// TIA Portal project "ENSACADORA_V4_021024_OPTIMIZADO" (V18)

(* hardware
DEVICE "SIMATIC 1200 station_1"  S7-1200 Station
   slot 0: "S7-1200 rack"  S7-1200 Rack  Rack  V1.0
   slot 1: "Master"  CPU 1212C DC/DC/Rly  6ES7 212-1HE40-0XB0  V4.5
   slot 2: "DI 8x24VDC/DQ 8xRelay_1"  SM 1223 DI8/DQ8 x relay  6ES7 223-1PH32-0XB0  V2.0
   slot 3: "AQ 2x14BIT_1"  SM 1232 AQ2  6ES7 232-4HB32-0XB0  V2.1
   slot 101: "CM 1241 (RS422/485)_1"  6ES7 241-1CH32-0XB0  V2.2
*)

// ===== PLC "Master"  CPU 1212C DC/DC/Rly =====

VAR_GLOBAL   // PLC tag table "A_Bits_programa"
   "COM_ACTIVA" AT %M261.1 : Bool;
   "AUX_OUT_VIBRADOR_TIME" AT %M267.1 : Bool;
   "ABRIENDO_COMP_CARGA" AT %M267.0 : Bool;
   "AUX_TIME_VIBRADOR" AT %M266.7 : Bool;
   "ACTIVAR MOTOR" AT %M266.6 : Bool;
   "AUX_OUT_COMPUERTA_BARRIDO_ABIERTA" AT %M266.5 : Bool;
   "AUX_OUT_VIBRADOR_BARRIDO" AT %M266.4 : Bool;
   "AUX_OUT_MOTOR_BARRIDO" AT %M266.3 : Bool;
   "AUX_OUT_COMPUERTA_MANUAL" AT %M266.2 : Bool;
   "AUX_OUT_VIBRADOR_MANUAL" AT %M266.1 : Bool;
   "AUX_OUT_MOTOR_MANUAL" AT %M266.0 : Bool;
   "ZERO RES" AT %M265.7 : Bool;
   "AUX_HACER_ZERO" AT %M265.6 : Bool;
   "BAS_EN_ZERO" AT %M265.5 : Bool;
   "BAS_TARA_HECHA" AT %M265.4 : Bool;
   "BAS_OVERLOAD" AT %M265.3 : Bool;
   "BAS_UNDERLOAD" AT %M265.2 : Bool;
   "BAS_ESTABLE" AT %M265.1 : Bool;
   "PB_POLARIDAD" AT %M265.0 : Bool;
   "AUX_SENSOR_COMP_CARGA_ABIERTA" AT %M264.7 : Bool;
   "AUX_VAL_COMP_CARGA_ABIERTA" AT %M264.6 : Bool;
   "AUX_INICIAR_CICLO" AT %M264.5 : Bool;
   "AUX_ERROR_COM_BASCULA" AT %M264.4 : Bool;
   "AUX_RESET_CICLO" AT %M264.3 : Bool;
   "AUX_MODO_BARRIDO" AT %M264.2 : Bool;
   "AUX_MODO_AUTOMATICO" AT %M264.1 : Bool;
   "AUX_MODO_MANUAL" AT %M264.0 : Bool;
   "AUX_INICIAR_LLENADO" AT %M256.0 : Bool;
   "AUX_PARAR_LLENADO" AT %M256.1 : Bool;
   "AUX_PARO_EMERGENCIA" AT %M256.2 : Bool;
   "AUX_SENSOR_INICIO_COMPUERTA" AT %M256.3 : Bool;
   "AUX_SENSOR_FINAL_COMPUERTA" AT %M256.4 : Bool;
   "FirstScan_PREGUNTAR" AT %M50.0 : Bool;
   "SENTIDO_MOTOR" AT %M259.3 : Bool;
   "AUX_ZERO_MANUAL" AT %M260.6 : Bool;
   "FrmHmi_HacerZeroBas" AT %M260.7 : Bool;
   "FrmHmi_ResetFallas" AT %M261.0 : Bool;   // x
   "RESETEAR FALLAS" AT %M261.2 : Bool;
   "INCIAR_CICLO" AT %M262.0 : Bool;
   "APAGAR_CICLO" AT %M262.1 : Bool;
   "AUX_INPUT_SOBRECARGA_MOTOR" AT %M262.6 : Bool;
   "AUX_FALLA_ARRANQUE_VDF" AT %M256.5 : Bool;
   "AUX_FALLA_COMPUERTA_ABIERTA_DOSIFICAR" AT %M256.6 : Bool;
   "AUX_FALLA_VARIADOR" AT %M256.7 : Bool;
   "AUX_BLINK_TORRETA_AMARILLO_ON" AT %M259.4 : Bool;
   "AUX_BLINK_TORRETA_AMARILLO_OFF" AT %M259.5 : Bool;
   "AUX_BLINK_TORRETA_VERDE_ON" AT %M259.6 : Bool;
   "AUX_BLINK_TORRETA_VERDE_OFF" AT %M259.7 : Bool;
   "AUX_OUT_TORRETA_C_ROJO" AT %M262.2 : Bool;
   "AUX_OUT_TORRETA_C_AMARILLO" AT %M262.3 : Bool;
   "AUX_OUT_TORRETA_C_VERDE" AT %M262.4 : Bool;
   "AUX_OUT_TORRETA_BUZZER" AT %M262.5 : Bool;
   "TOLERANCIA DE PESO BASCULA" AT %M259.0 : Bool;
   "SET_INDICADOR_CAPACIDAD" AT %M252.0 : Bool;
   "FROM_HMI_LEER_CAPACIDAD" AT %M252.1 : Bool;
   "PARO EMERGENCIA" AT %M252.2 : Bool;
END_VAR

VAR_GLOBAL   // PLC tag table "A_Byte_programa"
   "STEP_COM" AT %MB257 : Byte;
END_VAR

VAR_GLOBAL   // PLC tag table "A_Word_programa"
   "Refe_Frec_FromHmi_ToVdf_PENDENTE" AT %MW0 : Int;
   "SETPOINT" AT %MW2 : Int;
   "ESTATUS_OPERACION" AT %MW8 : Int;
   "STEP_BASCULA" AT %MW10 : Int;
   "ESTATUS VARIADOR" AT %MW268 : Word;
END_VAR

VAR_GLOBAL   // PLC tag table "A_DWord_programa"
   "TARAR" AT %MD36 : Real;
   "PESO_NETO" AT %MD40 : Real;
   "PESO_NETO_BASCULA" AT %MD44 : Real;
   "MAYOR_QUE_SETPOINT" AT %MD48 : Real;
   "MENOR_QUE_SETPOINT" AT %MD52 : Real;
   "DIV" AT %MD20 : DWord;
   "FILTRO" AT %MD24 : DWord;
   "DIFERENCIA" AT %MD28 : DWord;
   "PUNTO DE CORTE" AT %MD32 : DWord;
   "DEFAULT CORTE SETPOINT" AT %MD4 : DWord;
   "TOLERANCIA DE PESO MAXIMO" AT %MD272 : DWord;
   "PESO NETO BASCULA ENTERO" AT %MD276 : DWord;
   "SALIDA REF FREC DIVIDA HMI" AT %MD280 : DWord;
   "SALIDA FREC DIVIDIDA HMI" AT %MD284 : DWord;
   "lectura resgistro bascula" AT %MD56 : UDInt;
   "SALIDA AMPERAJE" AT %MD60 : Real;
END_VAR

VAR_GLOBAL   // PLC tag table "B_Calibracion"
   "ENVIAR_PESO_A_CALIBRAR" AT %M271.7 : Bool;
   "CONFIRMAR_PESO_CALIBRAR" AT %M271.6 : Bool;
   "CANCELAR_CALIBRACION" AT %M271.5 : Bool;
   "GUARDAR_CALIBRACION" AT %M271.4 : Bool;
   "CAPTURAR_PESO_BASCULA" AT %M271.3 : Bool;
   "CAPTURAR_ZERO_BASCULA" AT %M271.2 : Bool;
   "RESET_INDICADOR" AT %M271.1 : Bool;
   "VER_CALIBRACION" AT %M271.0 : Bool;
   "PESO_PARA_CALIBRAR" AT %MD92 : DInt;
END_VAR

VAR_GLOBAL   // PLC tag table "C_Fallas"
   "TIEMPO_APAGADO_VIBRADOR" AT %MD16 : DInt;
   "TIEMPO_ENCENDIDO_VIBRADOR" AT %MD12 : DInt;
   "Falla sobrecarga motor" AT %M270.7 : Bool;
   "Falla subcarga bascula" AT %M270.6 : Bool;
   "Falla sobrecarga bascula" AT %M270.5 : Bool;
   "FALLA_NO_SE_PUEDE_INICIAR_EN_ZERO" AT %M270.4 : Bool;
   "Fallas activas" AT %M270.3 : Bool;
   "Falla en el tiempo de vibrador" AT %M270.2 : Bool;
   "Falla al abrir compuerta descarga" AT %M270.1 : Bool;
   "Falla al cerrar compuerta descarga" AT %M270.0 : Bool;
   "TIMER_FALLAS_ON" AT %M259.2 : Bool;
   "TIMER_FALLAS_OFF" AT %M259.1 : Bool;
   "ERROR_MODBUS" AT %M267.2 : Bool;
   "AUX_ERROR_MODBUS" AT %M267.3 : Bool;
   "ERROR_VARIADOR" AT %M267.4 : Bool;
   "AUX_ERROR_VARIADOR" AT %M267.5 : Bool;
   "ERROR AL ENCENDER EL VARIADOR" AT %M267.6 : Bool;
   "FALLA AL ENCENDER EL MOTOR CON LA COMPUERTA CERRADA" AT %M267.7 : Bool;
END_VAR

VAR_GLOBAL   // PLC tag table "D_Entradas"
   "Input_SensorInicioPistonComp" AT %I0.4 : Bool;
   "Input_IniciarLLenado" AT %I0.0 : Bool;
   "Input_ParoEmergencia" AT %I0.2 : Bool;
   "Input_PararLLenado" AT %I0.1 : Bool;
   "Input_Sobrecarga_motor" AT %I0.3 : Bool;
   "Input_SensorFinPistonComp" AT %I0.5 : Bool;
END_VAR

VAR_GLOBAL   // PLC tag table "D_Salidas"
   "OUT_COMPUERTA_ABIERTA" AT %Q0.0 : Bool;
   "OUT_VIBRADOR" AT %Q0.1 : Bool;
   "TORRETA_C_ROJO" AT %Q0.3 : Bool;
   "TORRETA_C_AMARILLO" AT %Q0.4 : Bool;
   "TORRETA_C_VERDE" AT %Q0.5 : Bool;
   "TORRETA_BUZZER" AT %Q0.2 : Bool;
   "Kg_To_CCM" AT %QW112 : Word;
END_VAR

VAR_GLOBAL   // PLC tag table "E_Hmi"
   "FrmHmi_Barrido" AT %M263.4 : Bool;
   "FrmHmi_DesactivarModBarrido" AT %M263.3 : Bool;
   "FrmHmi_ActivarModBarrido" AT %M263.2 : Bool;
   "FrmHmi_Automatico" AT %M263.1 : Bool;
   "FrmHmi_ModManual" AT %M263.0 : Bool;
   "FrmHmi_ApagarVibradorEnsacadora" AT %M260.5 : Bool;
   "FrmHmi_EncenderVibradorEnsacadora" AT %M260.4 : Bool;
   "FrmHmi_DesactivarPistonCompuerta" AT %M260.3 : Bool;
   "FrmHmi_ActivarPistonCompuerta" AT %M260.2 : Bool;
   "FrmHmi_ApagarMotorHelicoidal" AT %M260.1 : Bool;
   "FrmHmi_EncenderMotorHelicoidal" AT %M260.0 : Bool;
END_VAR

TYPE "typeModbusCommLoad"
VERSION : 0.1
   STRUCT
      done : Bool := FALSE;
      error : Bool := FALSE;
      status : Word := W#16#0;
      errorStatus : Word := W#16#0;
      doneStored : Bool := FALSE;
   END_STRUCT;
END_TYPE

TYPE "typeModbusMaster"
VERSION : 0.1
   STRUCT
      req : Bool := FALSE;
      mbAddr : UInt;
      mode : USInt := 0;
      dataAddr : UDInt := 0;
      dataLen : UInt := 0;
      done : Bool := FALSE;
      busy : Bool := FALSE;
      error : Bool := FALSE;
      status : Word := W#16#0;
      errorStatus : Word := W#16#0;
   END_STRUCT;
END_TYPE

TYPE "typeDataPtr"
VERSION : 0.1
   STRUCT
      data : Array[0..11] of Int;
   END_STRUCT;
END_TYPE

TYPE "typeModbusVariador"
   STRUCT
      req : Bool := FALSE;
      mbAddr : UInt := 0;
      mode : USInt := 0;
      dataAddr : UDInt := 0;
      dataLen : UInt := 0;
      done : Bool := FALSE;
      busy : Bool := FALSE;
      error : Bool := FALSE;
      status : Word;
      errorStatus : Word;
   END_STRUCT;
END_TYPE

DATA_BLOCK "MasterData"   // DB1
{ S7_Optimized_Access := 'FALSE' }
VERSION : 0.1
   VAR
      "WRITE BASCULA" : Array[0..3] of Int;
      "READ BASCULA" : Array[0..10] of Int;
      "STATUS CAL" : Array[0..9] of Int;
      "WRITE VDF MOTOR" : Array[0..1] of Int;
      "READ VDF MOTOR" : Array[0..10] of Int;
      "PESO CALIBRAR" : Array[0..1] of Int;
      "LEER PESO CALIBRAR" : Array[0..2] of Int;
      "CAPACIDAD INDICADOR" : Array[0..1] of Int;
   END_VAR
BEGIN
END_DATA_BLOCK

DATA_BLOCK "Process"   // DB3
{ S7_Optimized_Access := 'TRUE' }
VERSION : 0.1
   VAR
      "step" : USInt := 1;
      edge : Bool := false;
      modbusMaster : "typeModbusMaster";
      modbusCommLoad : "typeModbusCommLoad";
   END_VAR
BEGIN
   modbusMaster.mbAddr := 2;
   modbusMaster.dataLen := 2;
END_DATA_BLOCK

DATA_BLOCK "HACER TARA_DB"   // DB6
{ S7_Optimized_Access := 'TRUE' }
VERSION : 0.1
// stored: InstanceOfName HACER TARA
"HACER TARA"
BEGIN
END_DATA_BLOCK

DATA_BLOCK "PORCENTAJE DE CORTE VDF GRUESO_DB_DB"   // DB9
{ S7_Optimized_Access := 'TRUE' }
VERSION : 0.1
// stored: InstanceOfName PORCENTAJE DE CORTE VDF GRUESO_DB
"PORCENTAJE DE CORTE VDF GRUESO_DB"
BEGIN
END_DATA_BLOCK

DATA_BLOCK "HACER TARA_DB_1"   // DB11
{ S7_Optimized_Access := 'TRUE' }
VERSION : 0.1
// stored: InstanceOfName HACER TARA
"HACER TARA"
BEGIN
END_DATA_BLOCK

DATA_BLOCK "db_variador"   // DB27
{ S7_Optimized_Access := 'TRUE' }
VERSION : 0.1
   VAR
      modbusVariador : "typeModbusVariador";
   END_VAR
BEGIN
END_DATA_BLOCK

// folder: System blocks/Program resources

DATA_BLOCK "IEC_Timer_0_DB"   // DB2
{ S7_Optimized_Access := 'TRUE' }
AUTHOR : Simatic
FAMILY : IEC
NAME : IEC_TMR
VERSION : 1.0
// stored: InstanceOfName IEC_TIMER
"IEC_TIMER"
BEGIN
END_DATA_BLOCK

DATA_BLOCK "IEC_Timer_0_DB_1"   // DB7
{ S7_Optimized_Access := 'TRUE' }
AUTHOR : Simatic
FAMILY : IEC
NAME : IEC_TMR
VERSION : 1.0
// stored: InstanceOfName IEC_TIMER
"IEC_TIMER"
BEGIN
END_DATA_BLOCK

DATA_BLOCK "IEC_Timer_0_DB_2"   // DB8
{ S7_Optimized_Access := 'TRUE' }
AUTHOR : Simatic
FAMILY : IEC
NAME : IEC_TMR
VERSION : 1.0
// stored: InstanceOfName IEC_TIMER
"IEC_TIMER"
BEGIN
END_DATA_BLOCK

DATA_BLOCK "IEC_Timer_0_DB_3"   // DB10
{ S7_Optimized_Access := 'TRUE' }
AUTHOR : Simatic
FAMILY : IEC
NAME : IEC_TMR
VERSION : 1.0
// stored: InstanceOfName IEC_TIMER
"IEC_TIMER"
BEGIN
END_DATA_BLOCK

DATA_BLOCK "IEC_Timer_0_DB_4"   // DB12
{ S7_Optimized_Access := 'TRUE' }
AUTHOR : Simatic
FAMILY : IEC
NAME : IEC_TMR
VERSION : 1.0
// stored: InstanceOfName IEC_TIMER
"IEC_TIMER"
BEGIN
END_DATA_BLOCK

DATA_BLOCK "IEC_Timer_0_DB_5"   // DB13
{ S7_Optimized_Access := 'TRUE' }
AUTHOR : Simatic
FAMILY : IEC
NAME : IEC_TMR
VERSION : 1.0
// stored: InstanceOfName IEC_TIMER
"IEC_TIMER"
BEGIN
END_DATA_BLOCK

DATA_BLOCK "IEC_Timer_0_DB_6"   // DB14
{ S7_Optimized_Access := 'TRUE' }
AUTHOR : Simatic
FAMILY : IEC
NAME : IEC_TMR
VERSION : 1.0
// stored: InstanceOfName IEC_TIMER
"IEC_TIMER"
BEGIN
END_DATA_BLOCK

DATA_BLOCK "IEC_Timer_0_DB_7"   // DB15
{ S7_Optimized_Access := 'TRUE' }
AUTHOR : Simatic
FAMILY : IEC
NAME : IEC_TMR
VERSION : 1.0
// stored: InstanceOfName IEC_TIMER
"IEC_TIMER"
BEGIN
END_DATA_BLOCK

DATA_BLOCK "IEC_Timer_0_DB_8"   // DB16
{ S7_Optimized_Access := 'TRUE' }
AUTHOR : Simatic
FAMILY : IEC
NAME : IEC_TMR
VERSION : 1.0
// stored: InstanceOfName IEC_TIMER
"IEC_TIMER"
BEGIN
END_DATA_BLOCK

DATA_BLOCK "IEC_Timer_0_DB_9"   // DB17
{ S7_Optimized_Access := 'TRUE' }
AUTHOR : Simatic
FAMILY : IEC
NAME : IEC_TMR
VERSION : 1.0
// stored: InstanceOfName IEC_TIMER
"IEC_TIMER"
BEGIN
END_DATA_BLOCK

DATA_BLOCK "IEC_Timer_0_DB_10"   // DB18
{ S7_Optimized_Access := 'TRUE' }
AUTHOR : Simatic
FAMILY : IEC
NAME : IEC_TMR
VERSION : 1.0
// stored: InstanceOfName IEC_TIMER
"IEC_TIMER"
BEGIN
END_DATA_BLOCK

DATA_BLOCK "IEC_Timer_0_DB_11"   // DB19
{ S7_Optimized_Access := 'TRUE' }
AUTHOR : Simatic
FAMILY : IEC
NAME : IEC_TMR
VERSION : 1.0
// stored: InstanceOfName IEC_TIMER
"IEC_TIMER"
BEGIN
END_DATA_BLOCK

DATA_BLOCK "IEC_Timer_0_DB_17"   // DB20
{ S7_Optimized_Access := 'TRUE' }
AUTHOR : Simatic
FAMILY : IEC
NAME : IEC_TMR
VERSION : 1.0
// stored: InstanceOfName IEC_TIMER
"IEC_TIMER"
BEGIN
END_DATA_BLOCK

DATA_BLOCK "IEC_Timer_0_DB_12"   // DB21
{ S7_Optimized_Access := 'TRUE' }
AUTHOR : Simatic
FAMILY : IEC
NAME : IEC_TMR
VERSION : 1.0
// stored: InstanceOfName IEC_TIMER
"IEC_TIMER"
BEGIN
END_DATA_BLOCK

DATA_BLOCK "IEC_Timer_0_DB_13"   // DB22
{ S7_Optimized_Access := 'TRUE' }
AUTHOR : Simatic
FAMILY : IEC
NAME : IEC_TMR
VERSION : 1.0
// stored: InstanceOfName IEC_TIMER
"IEC_TIMER"
BEGIN
END_DATA_BLOCK

DATA_BLOCK "IEC_Timer_0_DB_19"   // DB23
{ S7_Optimized_Access := 'TRUE' }
AUTHOR : Simatic
FAMILY : IEC
NAME : IEC_TMR
VERSION : 1.0
// stored: InstanceOfName IEC_TIMER
"IEC_TIMER"
BEGIN
END_DATA_BLOCK

DATA_BLOCK "IEC_Timer_0_DB_14"   // DB24
{ S7_Optimized_Access := 'TRUE' }
AUTHOR : Simatic
FAMILY : IEC
NAME : IEC_TMR
VERSION : 1.0
// stored: InstanceOfName IEC_TIMER
"IEC_TIMER"
BEGIN
END_DATA_BLOCK

DATA_BLOCK "IEC_Timer_0_DB_15"   // DB25
{ S7_Optimized_Access := 'TRUE' }
AUTHOR : Simatic
FAMILY : IEC
NAME : IEC_TMR
VERSION : 1.0
// stored: InstanceOfName IEC_TIMER
"IEC_TIMER"
BEGIN
END_DATA_BLOCK

DATA_BLOCK "IEC_Timer_0_DB_16"   // DB26
{ S7_Optimized_Access := 'TRUE' }
AUTHOR : Simatic
FAMILY : IEC
NAME : IEC_TMR
VERSION : 1.0
// stored: InstanceOfName IEC_TIMER
"IEC_TIMER"
BEGIN
END_DATA_BLOCK

DATA_BLOCK "IEC_Timer_0_DB_18"   // DB28
{ S7_Optimized_Access := 'TRUE' }
AUTHOR : Simatic
FAMILY : IEC
NAME : IEC_TMR
VERSION : 1.0
// stored: InstanceOfName IEC_TIMER
"IEC_TIMER"
BEGIN
END_DATA_BLOCK

DATA_BLOCK "IEC_Timer_0_DB_20"   // DB29
{ S7_Optimized_Access := 'TRUE' }
AUTHOR : Simatic
FAMILY : IEC
NAME : IEC_TMR
VERSION : 1.0
// stored: InstanceOfName IEC_TIMER
"IEC_TIMER"
BEGIN
END_DATA_BLOCK

// folder: (top level)

FUNCTION_BLOCK "HACER TARA"   // FB1, LAD
{ S7_Optimized_Access := 'TRUE' }
VERSION : 0.1
   VAR_INPUT
      TARAR2 : Bool;
      TARAR1 : Bool;
   END_VAR
   VAR_OUTPUT
      "PESO NETO TARA" : Real;
   END_VAR
   VAR_TEMP
      TARA : Real;
      TA : Bool;
      TA2 : Bool;
      available : Bool;
   END_VAR
   VAR_TEMP   // added for the SCL form of the ladder/FBD networks
      _w1 : Bool;
   END_VAR
BEGIN

REGION Network 1
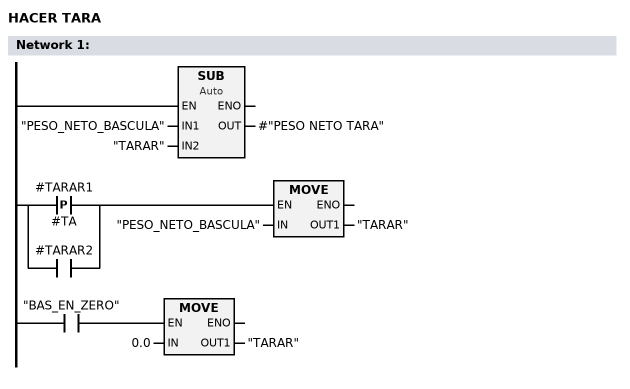
   RUNG wire#powerrail
      Sub(in1 := "PESO_NETO_BASCULA", in2 := "TARAR", out => #"PESO NETO TARA")
   END_RUNG
   RUNG wire#powerrail
      P_Contact(operand := #TARAR1, bit := #TA)
      wire#w1
      Move(in := "PESO_NETO_BASCULA", out1 => "TARAR")
   END_RUNG
   RUNG wire#powerrail
      Contact( #TARAR2 )
   END_RUNG wire#w1
   RUNG wire#powerrail
      Contact( "BAS_EN_ZERO" )
      Move(in := 0.0, out1 => "TARAR")
   END_RUNG
   // the same network as SCL:
   #"PESO NETO TARA" := "PESO_NETO_BASCULA" - "TARAR";
   #_w1 := #TARAR1 AND NOT #TA;   // rising edge of #TARAR1
   #TA := #TARAR1;
   IF #_w1 OR #TARAR2 THEN "TARAR" := "PESO_NETO_BASCULA"; END_IF;
   IF "BAS_EN_ZERO" THEN "TARAR" := 0.0; END_IF;
END_REGION
END_FUNCTION_BLOCK

FUNCTION_BLOCK "PORCENTAJE DE CORTE VDF GRUESO_DB"   // FB2, LAD
{ S7_Optimized_Access := 'TRUE' }
VERSION : 0.1
   VAR_INPUT
      "Set point" : Int;
      "% De Corte" : Int;
      PesoNeto : Real;
   END_VAR
   VAR_OUTPUT
      "Cantidad a cortar" : Real;
      "Bit OFF VDF Grueso" : Bool;
   END_VAR
   VAR_TEMP
      MULTI : Int;
   END_VAR
BEGIN

REGION Network 1
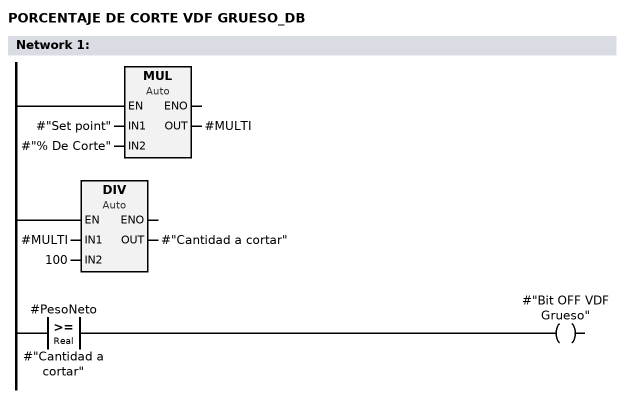
   RUNG wire#powerrail
      Mul(in1 := #"Set point", in2 := #"% De Corte", out => #MULTI)
   END_RUNG
   RUNG wire#powerrail
      Div(in1 := #MULTI, in2 := 100, out => #"Cantidad a cortar")
   END_RUNG
   RUNG wire#powerrail
      { S7_Templates := "SrcType := Real" } GE_Contact(in1 := #PesoNeto, in2 := #"Cantidad a cortar")
      Coil( #"Bit OFF VDF Grueso" )
   END_RUNG
   // the same network as SCL:
   #MULTI := #"Set point" * #"% De Corte";
   #"Cantidad a cortar" := #MULTI / 100;
   #"Bit OFF VDF Grueso" := #PesoNeto >= #"Cantidad a cortar";
END_REGION
END_FUNCTION_BLOCK

ORGANIZATION_BLOCK "1- COMUNICACION MODBUS"   // OB1, LAD, ProgramCycle
{ S7_Optimized_Access := 'TRUE' }
VERSION : 0.1
   VAR_INPUT
      Initial_Call : Bool;
      Remanence : Bool;
   END_VAR
   VAR_TEMP
      OutFrecMot : Int;
      OutRefFrecMot : Int;
      OutCorrienteMot : Real;
      "Bits Bascula" : DInt;
      "eroor com" : Bool;
      "weig neto" : Real;
      frecuencia : DInt;
   END_VAR
   VAR_TEMP   // added for the SCL form of the ladder/FBD networks
      _w1 : Bool;
   END_VAR
BEGIN

REGION Network 1: INICIALIZAR COMUNICACION
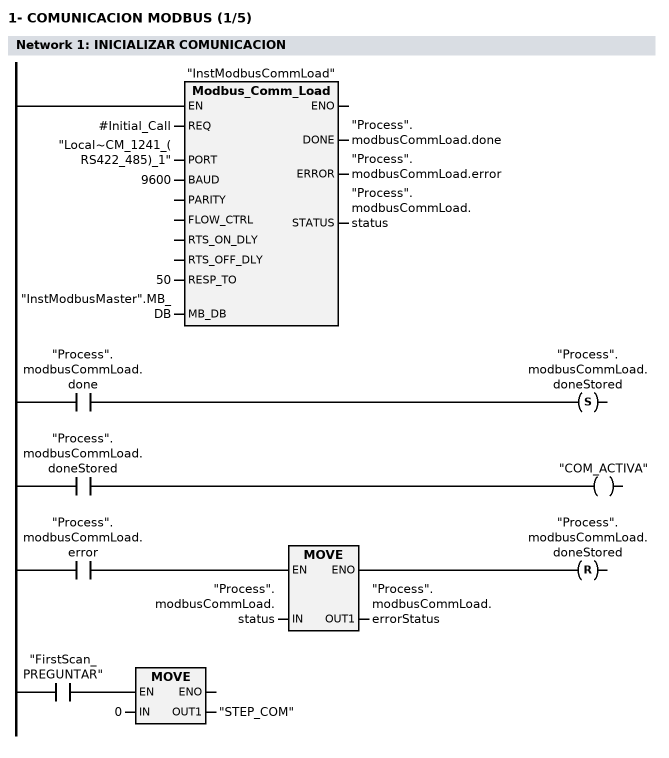
   // ENO of a box is taken as its EN; it also drops when the box reports an error
   "InstModbusCommLoad"(REQ := #Initial_Call,   // Modbus_Comm_Load
                        PORT := "Local~CM_1241_(RS422_485)_1",
                        BAUD := 9600,
                        RESP_TO := 50,
                        MB_DB := "InstModbusMaster".MB_DB,
                        DONE => "Process".modbusCommLoad.done,
                        ERROR => "Process".modbusCommLoad.error,
                        STATUS => "Process".modbusCommLoad.status);
   IF "Process".modbusCommLoad.done THEN "Process".modbusCommLoad.doneStored := TRUE; END_IF;
   "COM_ACTIVA" := "Process".modbusCommLoad.doneStored;
   IF "Process".modbusCommLoad.error THEN
       "Process".modbusCommLoad.errorStatus := "Process".modbusCommLoad.status;
       "Process".modbusCommLoad.doneStored := FALSE;
   END_IF;
   IF "FirstScan_PREGUNTAR" THEN "STEP_COM" := 0; END_IF;
END_REGION

REGION Network 2: LEER--ESCRIBIR, BASCULA
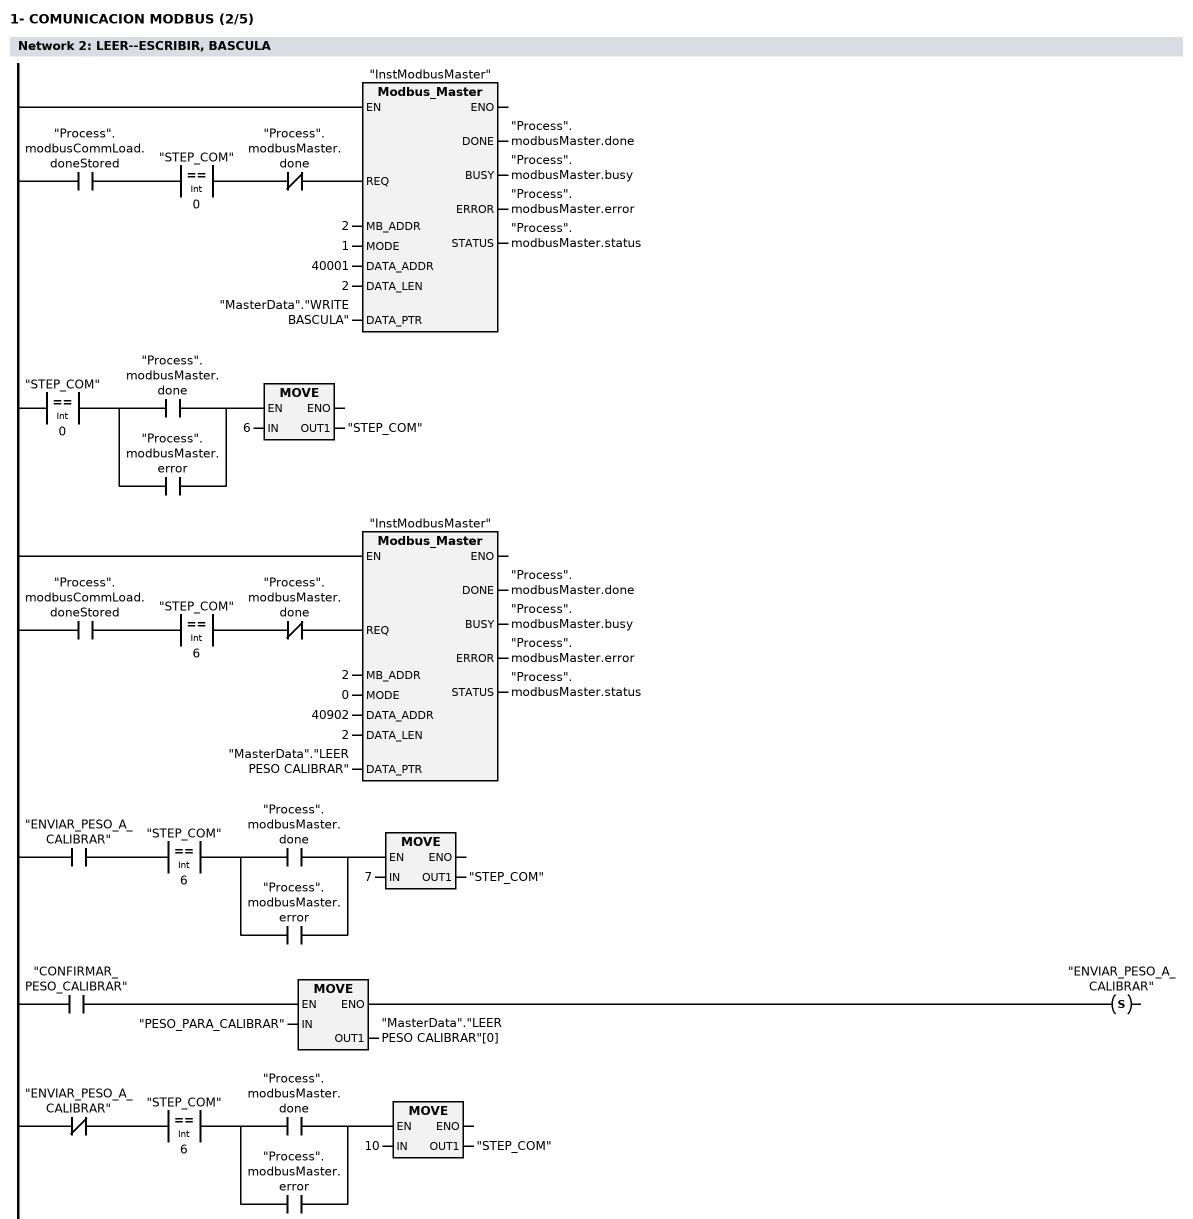
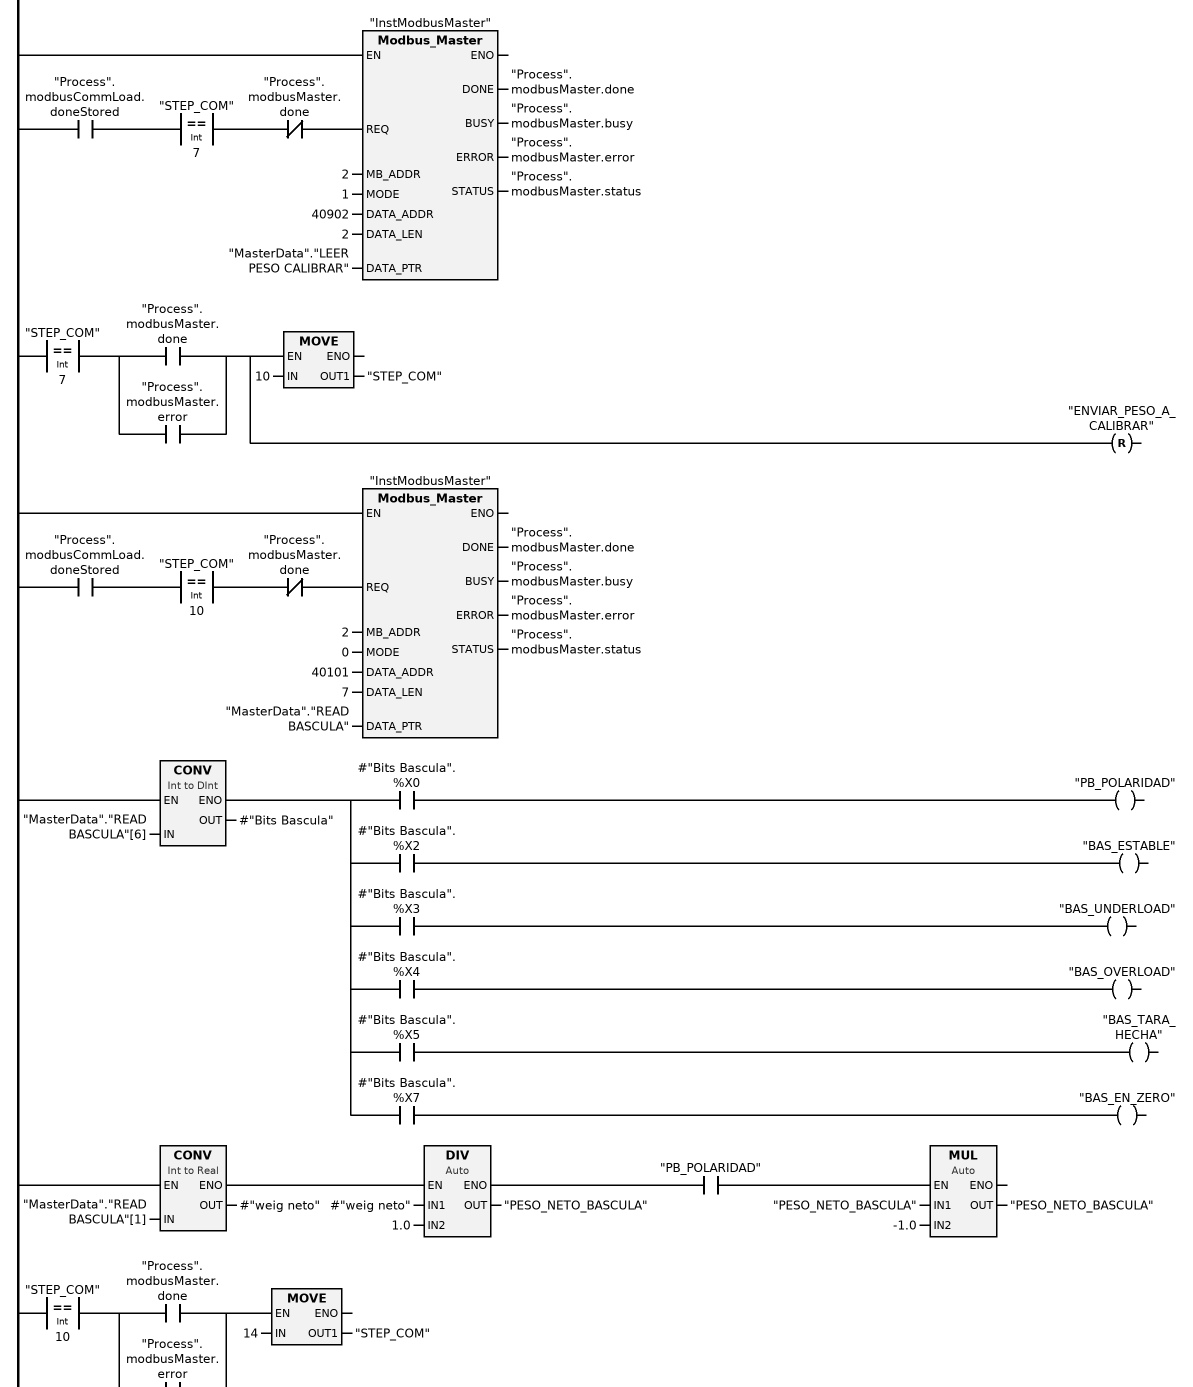
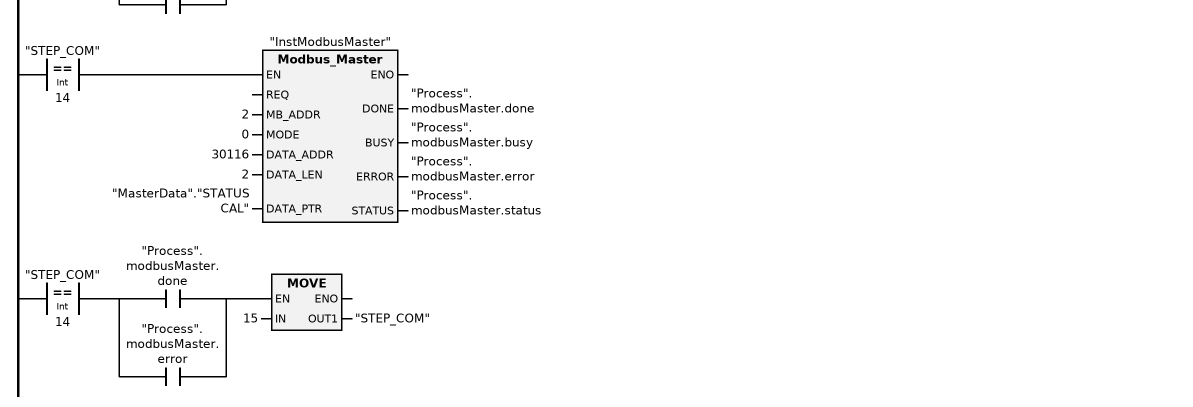
   "InstModbusMaster"(REQ := "Process".modbusCommLoad.doneStored AND ("STEP_COM" = 0) AND NOT "Process".modbusMaster.done,   // Modbus_Master
                      MB_ADDR := 2,
                      MODE := 1,
                      DATA_ADDR := 40001,
                      DATA_LEN := 2,
                      DATA_PTR := "MasterData"."WRITE BASCULA",
                      DONE => "Process".modbusMaster.done,
                      BUSY => "Process".modbusMaster.busy,
                      ERROR => "Process".modbusMaster.error,
                      STATUS => "Process".modbusMaster.status);
   IF ("STEP_COM" = 0) AND ("Process".modbusMaster.done OR "Process".modbusMaster.error) THEN
       "STEP_COM" := 6;
   END_IF;
   "InstModbusMaster"(REQ := "Process".modbusCommLoad.doneStored AND ("STEP_COM" = 6) AND NOT "Process".modbusMaster.done,   // Modbus_Master
                      MB_ADDR := 2,
                      MODE := 0,
                      DATA_ADDR := 40902,
                      DATA_LEN := 2,
                      DATA_PTR := "MasterData"."LEER PESO CALIBRAR",
                      DONE => "Process".modbusMaster.done,
                      BUSY => "Process".modbusMaster.busy,
                      ERROR => "Process".modbusMaster.error,
                      STATUS => "Process".modbusMaster.status);
   IF "ENVIAR_PESO_A_CALIBRAR" AND ("STEP_COM" = 6) AND ("Process".modbusMaster.done OR "Process".modbusMaster.error) THEN
       "STEP_COM" := 7;
   END_IF;
   IF "CONFIRMAR_PESO_CALIBRAR" THEN
       "MasterData"."LEER PESO CALIBRAR"[0] := "PESO_PARA_CALIBRAR";
       "ENVIAR_PESO_A_CALIBRAR" := TRUE;
   END_IF;
   IF NOT "ENVIAR_PESO_A_CALIBRAR" AND ("STEP_COM" = 6) AND ("Process".modbusMaster.done OR "Process".modbusMaster.error) THEN
       "STEP_COM" := 10;
   END_IF;
   "InstModbusMaster"(REQ := "Process".modbusCommLoad.doneStored AND ("STEP_COM" = 7) AND NOT "Process".modbusMaster.done,   // Modbus_Master
                      MB_ADDR := 2,
                      MODE := 1,
                      DATA_ADDR := 40902,
                      DATA_LEN := 2,
                      DATA_PTR := "MasterData"."LEER PESO CALIBRAR",
                      DONE => "Process".modbusMaster.done,
                      BUSY => "Process".modbusMaster.busy,
                      ERROR => "Process".modbusMaster.error,
                      STATUS => "Process".modbusMaster.status);
   #_w1 := ("STEP_COM" = 7) AND ("Process".modbusMaster.done OR "Process".modbusMaster.error);
   IF #_w1 THEN
       "STEP_COM" := 10;
       "ENVIAR_PESO_A_CALIBRAR" := FALSE;
   END_IF;
   "InstModbusMaster"(REQ := "Process".modbusCommLoad.doneStored AND ("STEP_COM" = 10) AND NOT "Process".modbusMaster.done,   // Modbus_Master
                      MB_ADDR := 2,
                      MODE := 0,
                      DATA_ADDR := 40101,
                      DATA_LEN := 7,
                      DATA_PTR := "MasterData"."READ BASCULA",
                      DONE => "Process".modbusMaster.done,
                      BUSY => "Process".modbusMaster.busy,
                      ERROR => "Process".modbusMaster.error,
                      STATUS => "Process".modbusMaster.status);
   #"Bits Bascula" := INT_TO_DINT("MasterData"."READ BASCULA"[6]);
   "PB_POLARIDAD" := #"Bits Bascula".%X0;
   "BAS_ESTABLE" := #"Bits Bascula".%X2;
   "BAS_UNDERLOAD" := #"Bits Bascula".%X3;
   "BAS_OVERLOAD" := #"Bits Bascula".%X4;
   "BAS_TARA_HECHA" := #"Bits Bascula".%X5;
   "BAS_EN_ZERO" := #"Bits Bascula".%X7;
   #"weig neto" := INT_TO_REAL("MasterData"."READ BASCULA"[1]);
   "PESO_NETO_BASCULA" := #"weig neto" / 1.0;
   IF "PB_POLARIDAD" THEN "PESO_NETO_BASCULA" := "PESO_NETO_BASCULA" * (-1.0); END_IF;
   IF ("STEP_COM" = 10) AND ("Process".modbusMaster.done OR "Process".modbusMaster.error) THEN
       "STEP_COM" := 14;
   END_IF;
   IF "STEP_COM" = 14 THEN
       "InstModbusMaster"(MB_ADDR := 2,   // Modbus_Master
                          MODE := 0,
                          DATA_ADDR := 30116,
                          DATA_LEN := 2,
                          DATA_PTR := "MasterData"."STATUS CAL",
                          DONE => "Process".modbusMaster.done,
                          BUSY => "Process".modbusMaster.busy,
                          ERROR => "Process".modbusMaster.error,
                          STATUS => "Process".modbusMaster.status);
   END_IF;
   IF ("STEP_COM" = 14) AND ("Process".modbusMaster.done OR "Process".modbusMaster.error) THEN
       "STEP_COM" := 15;
   END_IF;
END_REGION

REGION Network 3: FALLA EN LA BASCULA
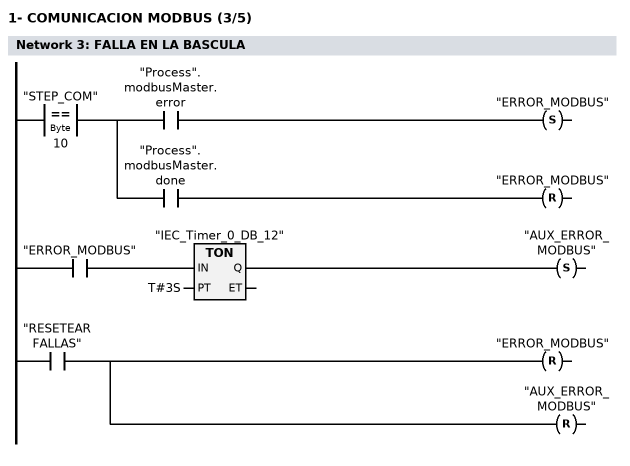
   #_w1 := "STEP_COM" = 10;
   IF #_w1 AND "Process".modbusMaster.error THEN "ERROR_MODBUS" := TRUE; END_IF;
   IF #_w1 AND "Process".modbusMaster.done THEN "ERROR_MODBUS" := FALSE; END_IF;
   "IEC_Timer_0_DB_12".TON(IN := "ERROR_MODBUS", PT := T#3S);
   IF "IEC_Timer_0_DB_12".Q THEN "AUX_ERROR_MODBUS" := TRUE; END_IF;
   IF "RESETEAR FALLAS" THEN
       "ERROR_MODBUS" := FALSE;
       "AUX_ERROR_MODBUS" := FALSE;
   END_IF;
END_REGION

REGION Network 4: LEER--ESCRIBIR, VDF MOTOR
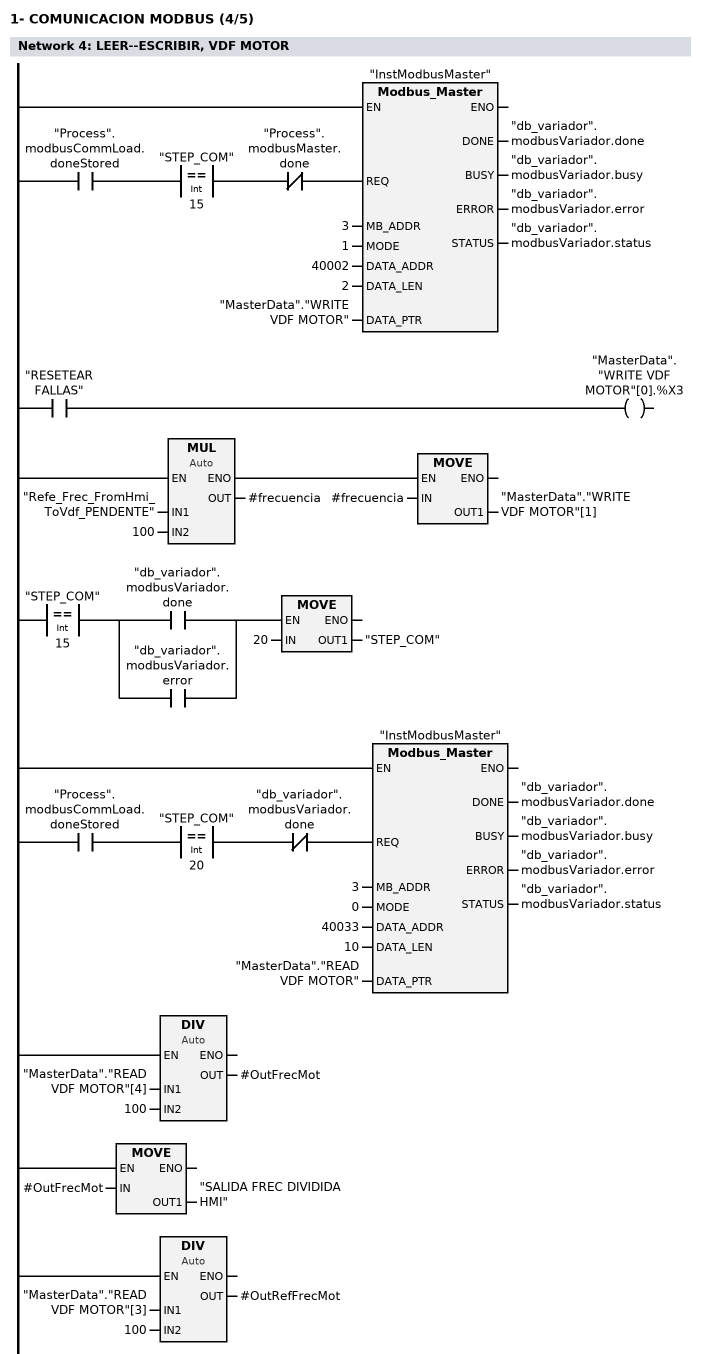
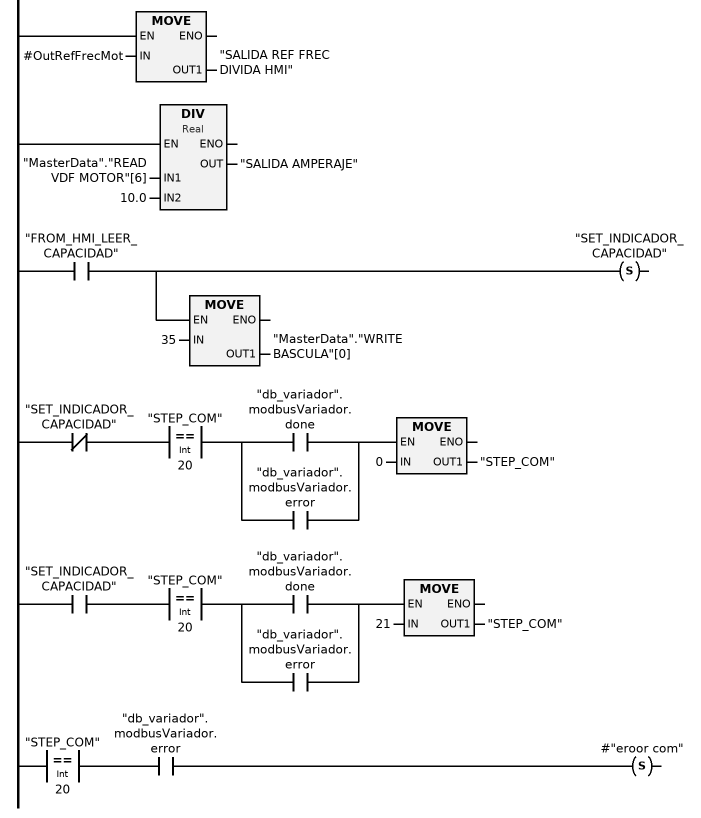
   "InstModbusMaster"(REQ := "Process".modbusCommLoad.doneStored AND ("STEP_COM" = 15) AND NOT "Process".modbusMaster.done,   // Modbus_Master
                      MB_ADDR := 3,
                      MODE := 1,
                      DATA_ADDR := 40002,
                      DATA_LEN := 2,
                      DATA_PTR := "MasterData"."WRITE VDF MOTOR",
                      DONE => "db_variador".modbusVariador.done,
                      BUSY => "db_variador".modbusVariador.busy,
                      ERROR => "db_variador".modbusVariador.error,
                      STATUS => "db_variador".modbusVariador.status);
   "MasterData"."WRITE VDF MOTOR"[0].%X3 := "RESETEAR FALLAS";
   #frecuencia := "Refe_Frec_FromHmi_ToVdf_PENDENTE" * 100;
   "MasterData"."WRITE VDF MOTOR"[1] := #frecuencia;
   IF ("STEP_COM" = 15) AND ("db_variador".modbusVariador.done OR "db_variador".modbusVariador.error) THEN
       "STEP_COM" := 20;
   END_IF;
   "InstModbusMaster"(REQ := "Process".modbusCommLoad.doneStored AND ("STEP_COM" = 20) AND NOT "db_variador".modbusVariador.done,   // Modbus_Master
                      MB_ADDR := 3,
                      MODE := 0,
                      DATA_ADDR := 40033,
                      DATA_LEN := 10,
                      DATA_PTR := "MasterData"."READ VDF MOTOR",
                      DONE => "db_variador".modbusVariador.done,
                      BUSY => "db_variador".modbusVariador.busy,
                      ERROR => "db_variador".modbusVariador.error,
                      STATUS => "db_variador".modbusVariador.status);
   #OutFrecMot := "MasterData"."READ VDF MOTOR"[4] / 100;
   "SALIDA FREC DIVIDIDA HMI" := #OutFrecMot;
   #OutRefFrecMot := "MasterData"."READ VDF MOTOR"[3] / 100;
   "SALIDA REF FREC DIVIDA HMI" := #OutRefFrecMot;
   "SALIDA AMPERAJE" := "MasterData"."READ VDF MOTOR"[6] / 10.0;
   IF "FROM_HMI_LEER_CAPACIDAD" THEN
       "SET_INDICADOR_CAPACIDAD" := TRUE;
       "MasterData"."WRITE BASCULA"[0] := 35;
   END_IF;
   IF NOT "SET_INDICADOR_CAPACIDAD" AND ("STEP_COM" = 20) AND ("db_variador".modbusVariador.done OR "db_variador".modbusVariador.error) THEN
       "STEP_COM" := 0;
   END_IF;
   IF "SET_INDICADOR_CAPACIDAD" AND ("STEP_COM" = 20) AND ("db_variador".modbusVariador.done OR "db_variador".modbusVariador.error) THEN
       "STEP_COM" := 21;
   END_IF;
   IF ("STEP_COM" = 20) AND "db_variador".modbusVariador.error THEN #"eroor com" := TRUE; END_IF;
END_REGION

REGION Network 5: LEER CAPACIDA DE BASCULA PARA CONVERSION 4MA-20MA A CMM
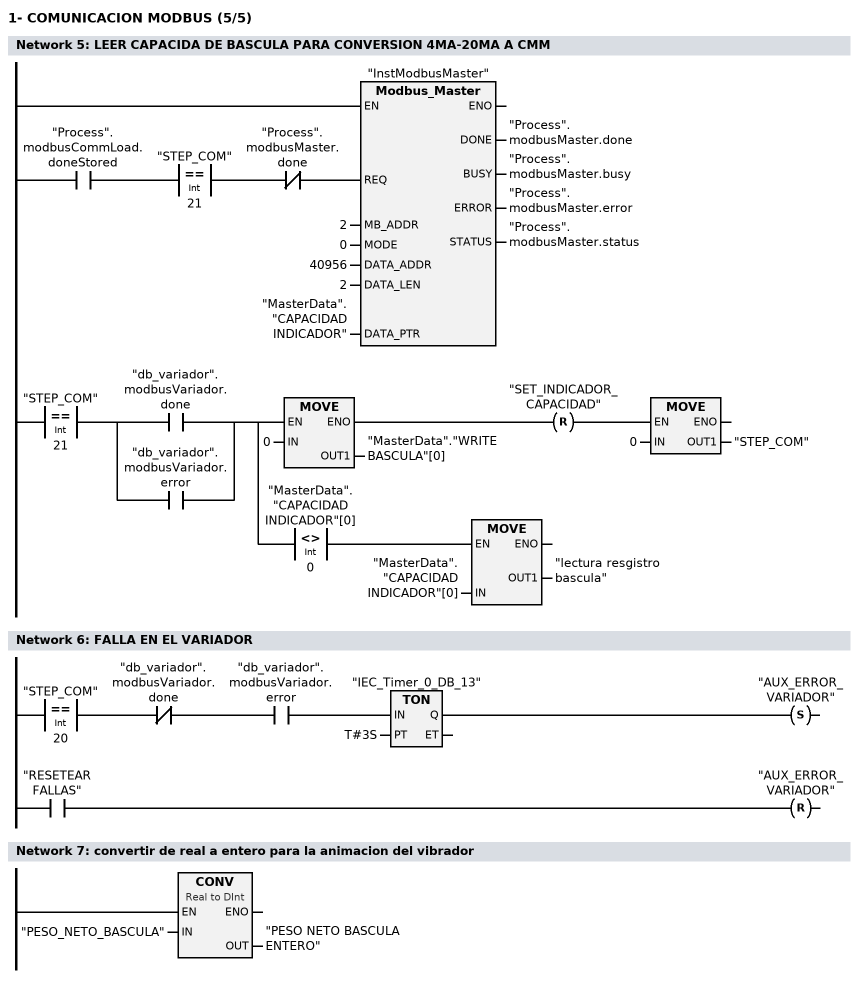
   "InstModbusMaster"(REQ := "Process".modbusCommLoad.doneStored AND ("STEP_COM" = 21) AND NOT "Process".modbusMaster.done,   // Modbus_Master
                      MB_ADDR := 2,
                      MODE := 0,
                      DATA_ADDR := 40956,
                      DATA_LEN := 2,
                      DATA_PTR := "MasterData"."CAPACIDAD INDICADOR",
                      DONE => "Process".modbusMaster.done,
                      BUSY => "Process".modbusMaster.busy,
                      ERROR => "Process".modbusMaster.error,
                      STATUS => "Process".modbusMaster.status);
   #_w1 := ("STEP_COM" = 21) AND ("db_variador".modbusVariador.done OR "db_variador".modbusVariador.error);
   IF #_w1 THEN
       "MasterData"."WRITE BASCULA"[0] := 0;
       "SET_INDICADOR_CAPACIDAD" := FALSE;
       "STEP_COM" := 0;
   END_IF;
   IF #_w1 AND ("MasterData"."CAPACIDAD INDICADOR"[0] <> 0) THEN
       "lectura resgistro bascula" := "MasterData"."CAPACIDAD INDICADOR"[0];
   END_IF;
END_REGION

REGION Network 6: FALLA EN EL VARIADOR
   "IEC_Timer_0_DB_13".TON(IN := ("STEP_COM" = 20) AND NOT "db_variador".modbusVariador.done AND "db_variador".modbusVariador.error,
                           PT := T#3S);
   IF "IEC_Timer_0_DB_13".Q THEN "AUX_ERROR_VARIADOR" := TRUE; END_IF;
   IF "RESETEAR FALLAS" THEN "AUX_ERROR_VARIADOR" := FALSE; END_IF;
END_REGION

REGION Network 7: convertir de real a entero para la animacion del vibrador
   RUNG wire#powerrail
      { S7_Templates := "[SrcType := Real, DestType := DInt]" } Convert(in := "PESO_NETO_BASCULA", out => "PESO NETO BASCULA ENTERO")
   END_RUNG
   // the same network as SCL:
   "PESO NETO BASCULA ENTERO" := REAL_TO_DINT("PESO_NETO_BASCULA");
END_REGION
END_ORGANIZATION_BLOCK

ORGANIZATION_BLOCK "2- ENTRADAS"   // OB123, LAD, ProgramCycle
{ S7_Optimized_Access := 'TRUE' }
VERSION : 0.1
   VAR_INPUT
      Initial_Call : Bool;
      Remanence : Bool;
   END_VAR
BEGIN

REGION Network 1: ENTRADAS FÍSICAS
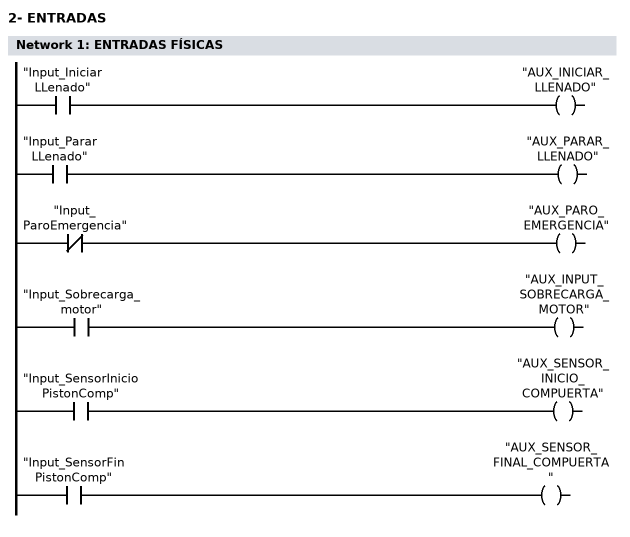
   RUNG wire#powerrail
      Contact( "Input_IniciarLLenado" )
      Coil( "AUX_INICIAR_LLENADO" )
   END_RUNG
   RUNG wire#powerrail
      Contact( "Input_PararLLenado" )
      Coil( "AUX_PARAR_LLENADO" )
   END_RUNG
   RUNG wire#powerrail
      I_Contact( "Input_ParoEmergencia" )
      Coil( "AUX_PARO_EMERGENCIA" )
   END_RUNG
   RUNG wire#powerrail
      Contact( "Input_Sobrecarga_motor" )
      Coil( "AUX_INPUT_SOBRECARGA_MOTOR" )
   END_RUNG
   RUNG wire#powerrail
      Contact( "Input_SensorInicioPistonComp" )
      Coil( "AUX_SENSOR_INICIO_COMPUERTA" )
   END_RUNG
   RUNG wire#powerrail
      Contact( "Input_SensorFinPistonComp" )
      Coil( "AUX_SENSOR_FINAL_COMPUERTA" )
   END_RUNG
   // the same network as SCL:
   "AUX_INICIAR_LLENADO" := "Input_IniciarLLenado";
   "AUX_PARAR_LLENADO" := "Input_PararLLenado";
   "AUX_PARO_EMERGENCIA" := NOT "Input_ParoEmergencia";
   "AUX_INPUT_SOBRECARGA_MOTOR" := "Input_Sobrecarga_motor";
   "AUX_SENSOR_INICIO_COMPUERTA" := "Input_SensorInicioPistonComp";
   "AUX_SENSOR_FINAL_COMPUERTA" := "Input_SensorFinPistonComp";
END_REGION
END_ORGANIZATION_BLOCK

ORGANIZATION_BLOCK "3- LOGICA LLENADO"   // OB124, LAD, ProgramCycle
{ S7_Optimized_Access := 'TRUE' }
VERSION : 0.1
   VAR_INPUT
      Initial_Call : Bool;
      Remanence : Bool;
   END_VAR
   VAR_TEMP
      inhabilitar : Bool;
      AVAILABLE : Bool;
      frecoMOT : Int;
      "TIME ENCENDIDO" : Time;
      "TIME APAGADO" : Time;
      "RESULTADO ENCENDIDO" : Int;
      "RESULTADO APAGADO" : Int;
      status_operacion : Bool;
   END_VAR
   VAR_TEMP   // added for the SCL form of the ladder/FBD networks
      _w1 : Bool;
      _w2 : Bool;
   END_VAR
BEGIN

REGION Network 1: MODO MANUAL, AUTOMATICO, BARRIDO
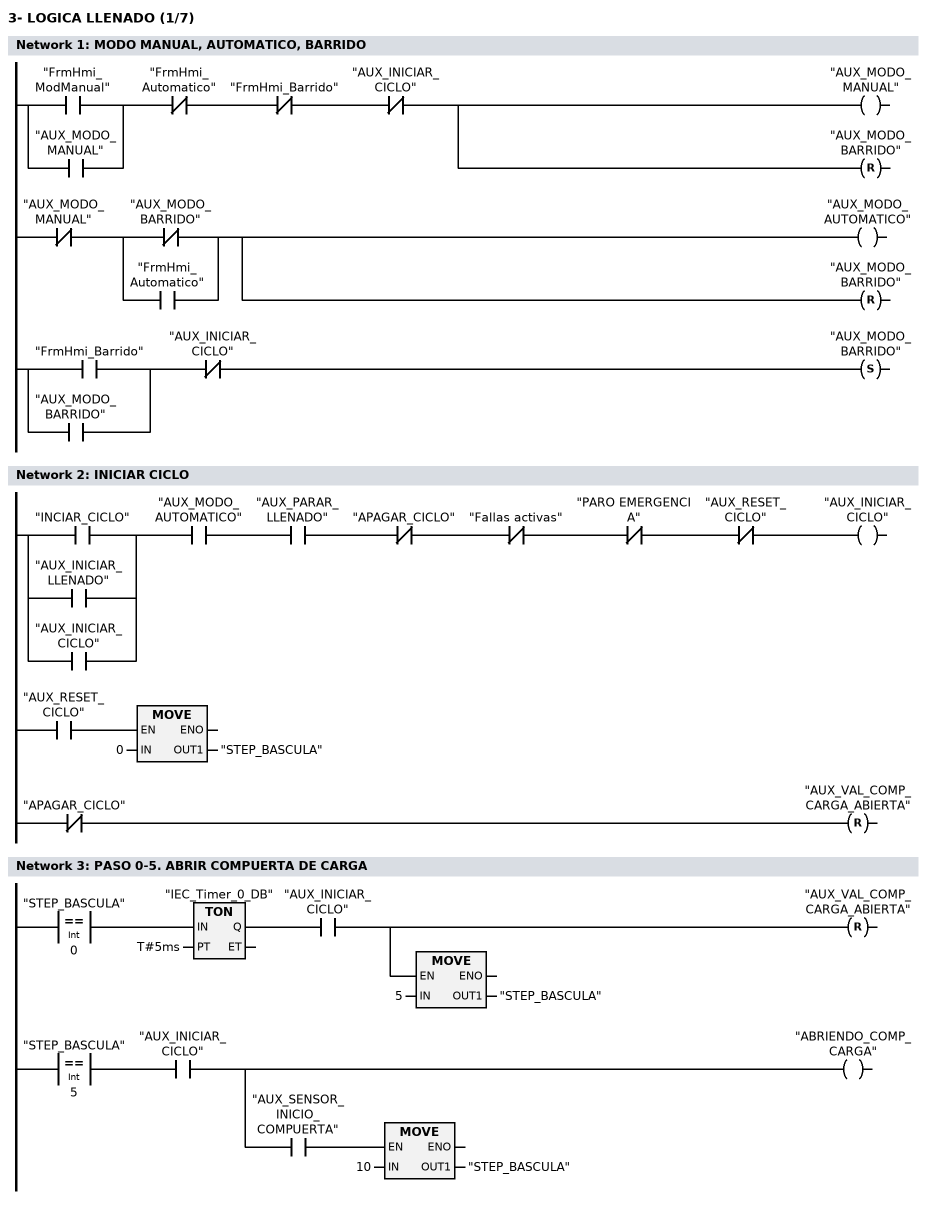
   RUNG wire#powerrail
      Contact( "FrmHmi_ModManual" )
      wire#w1
      I_Contact( "FrmHmi_Automatico" )
      I_Contact( "FrmHmi_Barrido" )
      I_Contact( "AUX_INICIAR_CICLO" )
      wire#w2
      Coil( "AUX_MODO_MANUAL" )
   END_RUNG
   RUNG wire#powerrail
      Contact( "AUX_MODO_MANUAL" )
   END_RUNG wire#w1
   RUNG wire#w2
      R_Coil( "AUX_MODO_BARRIDO" )
   END_RUNG
   RUNG wire#powerrail
      I_Contact( "AUX_MODO_MANUAL" )
      wire#w3
      I_Contact( "AUX_MODO_BARRIDO" )
      wire#w4
      Coil( "AUX_MODO_AUTOMATICO" )
   END_RUNG
   RUNG wire#w3
      Contact( "FrmHmi_Automatico" )
   END_RUNG wire#w4
   RUNG wire#w4
      R_Coil( "AUX_MODO_BARRIDO" )
   END_RUNG
   RUNG wire#powerrail
      Contact( "FrmHmi_Barrido" )
      wire#w5
      I_Contact( "AUX_INICIAR_CICLO" )
      S_Coil( "AUX_MODO_BARRIDO" )
   END_RUNG
   RUNG wire#powerrail
      Contact( "AUX_MODO_BARRIDO" )
   END_RUNG wire#w5
   // the same network as SCL:
   "AUX_MODO_MANUAL" := ("FrmHmi_ModManual" OR "AUX_MODO_MANUAL") AND NOT "FrmHmi_Automatico" AND NOT "FrmHmi_Barrido" AND NOT "AUX_INICIAR_CICLO";
   IF "AUX_MODO_MANUAL" THEN "AUX_MODO_BARRIDO" := FALSE; END_IF;
   "AUX_MODO_AUTOMATICO" := NOT "AUX_MODO_MANUAL" AND (NOT "AUX_MODO_BARRIDO" OR "FrmHmi_Automatico");
   IF "AUX_MODO_AUTOMATICO" THEN "AUX_MODO_BARRIDO" := FALSE; END_IF;
   IF ("FrmHmi_Barrido" OR "AUX_MODO_BARRIDO") AND NOT "AUX_INICIAR_CICLO" THEN
       "AUX_MODO_BARRIDO" := TRUE;
   END_IF;
END_REGION

REGION Network 2: INICIAR CICLO
   RUNG wire#powerrail
      Contact( "INCIAR_CICLO" )
      wire#w1
      Contact( "AUX_MODO_AUTOMATICO" )
      Contact( "AUX_PARAR_LLENADO" )
      I_Contact( "APAGAR_CICLO" )
      I_Contact( "Fallas activas" )
      I_Contact( "PARO EMERGENCIA" )
      I_Contact( "AUX_RESET_CICLO" )
      Coil( "AUX_INICIAR_CICLO" )
   END_RUNG
   RUNG wire#powerrail
      Contact( "AUX_INICIAR_LLENADO" )
   END_RUNG wire#w1
   RUNG wire#powerrail
      Contact( "AUX_INICIAR_CICLO" )
   END_RUNG wire#w1
   RUNG wire#powerrail
      Contact( "AUX_RESET_CICLO" )
      Move(in := 0, out1 => "STEP_BASCULA")
   END_RUNG
   RUNG wire#powerrail
      I_Contact( "APAGAR_CICLO" )
      R_Coil( "AUX_VAL_COMP_CARGA_ABIERTA" )
   END_RUNG
   // the same network as SCL:
   "AUX_INICIAR_CICLO" := ("INCIAR_CICLO" OR "AUX_INICIAR_LLENADO" OR "AUX_INICIAR_CICLO") AND "AUX_MODO_AUTOMATICO" AND "AUX_PARAR_LLENADO" AND NOT "APAGAR_CICLO" AND NOT "Fallas activas" AND NOT "PARO EMERGENCIA" AND NOT "AUX_RESET_CICLO";
   IF "AUX_RESET_CICLO" THEN "STEP_BASCULA" := 0; END_IF;
   IF NOT "APAGAR_CICLO" THEN "AUX_VAL_COMP_CARGA_ABIERTA" := FALSE; END_IF;
END_REGION

REGION Network 3: PASO 0-5. ABRIR COMPUERTA DE CARGA
   "IEC_Timer_0_DB".TON(IN := "STEP_BASCULA" = 0, PT := T#5ms);
   IF "IEC_Timer_0_DB".Q AND "AUX_INICIAR_CICLO" THEN
       "AUX_VAL_COMP_CARGA_ABIERTA" := FALSE;
       "STEP_BASCULA" := 5;
   END_IF;
   "ABRIENDO_COMP_CARGA" := ("STEP_BASCULA" = 5) AND "AUX_INICIAR_CICLO";
   IF "ABRIENDO_COMP_CARGA" AND "AUX_SENSOR_INICIO_COMPUERTA" THEN "STEP_BASCULA" := 10; END_IF;
END_REGION

REGION Network 4: PASO 10. HACER TARA
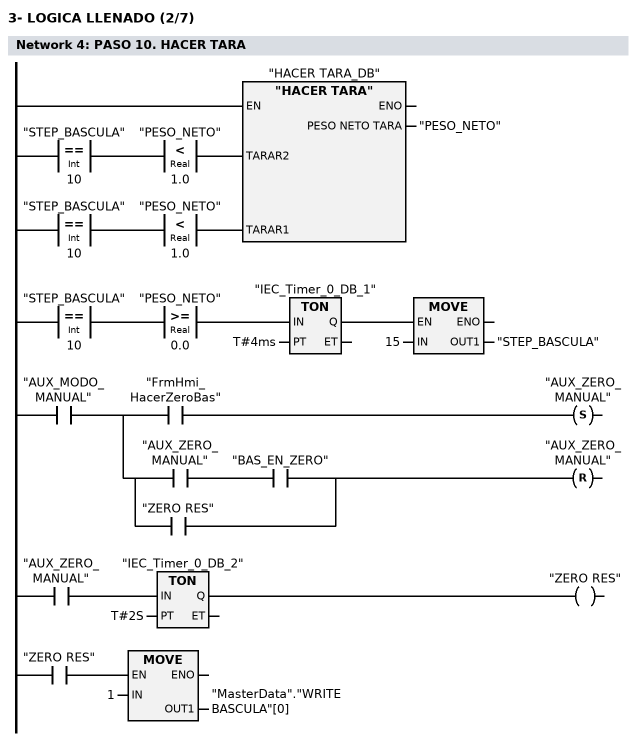
   "HACER TARA_DB"(TARAR2 := ("STEP_BASCULA" = 10) AND ("PESO_NETO" < 1.0),   // "HACER TARA"
                   TARAR1 := ("STEP_BASCULA" = 10) AND ("PESO_NETO" < 1.0),
                   "PESO NETO TARA" => "PESO_NETO");
   "IEC_Timer_0_DB_1".TON(IN := ("STEP_BASCULA" = 10) AND ("PESO_NETO" >= 0.0), PT := T#4ms);
   IF "IEC_Timer_0_DB_1".Q THEN "STEP_BASCULA" := 15; END_IF;
   IF "AUX_MODO_MANUAL" AND "FrmHmi_HacerZeroBas" THEN "AUX_ZERO_MANUAL" := TRUE; END_IF;
   IF "AUX_MODO_MANUAL" AND (("AUX_ZERO_MANUAL" AND "BAS_EN_ZERO") OR "ZERO RES") THEN
       "AUX_ZERO_MANUAL" := FALSE;
   END_IF;
   "IEC_Timer_0_DB_2".TON(IN := "AUX_ZERO_MANUAL", PT := T#2S);
   "ZERO RES" := "IEC_Timer_0_DB_2".Q;
   IF "ZERO RES" THEN "MasterData"."WRITE BASCULA"[0] := 1; END_IF;
END_REGION

REGION Network 5: PASO 15. ENCENDER Y APAGAR MOTORES
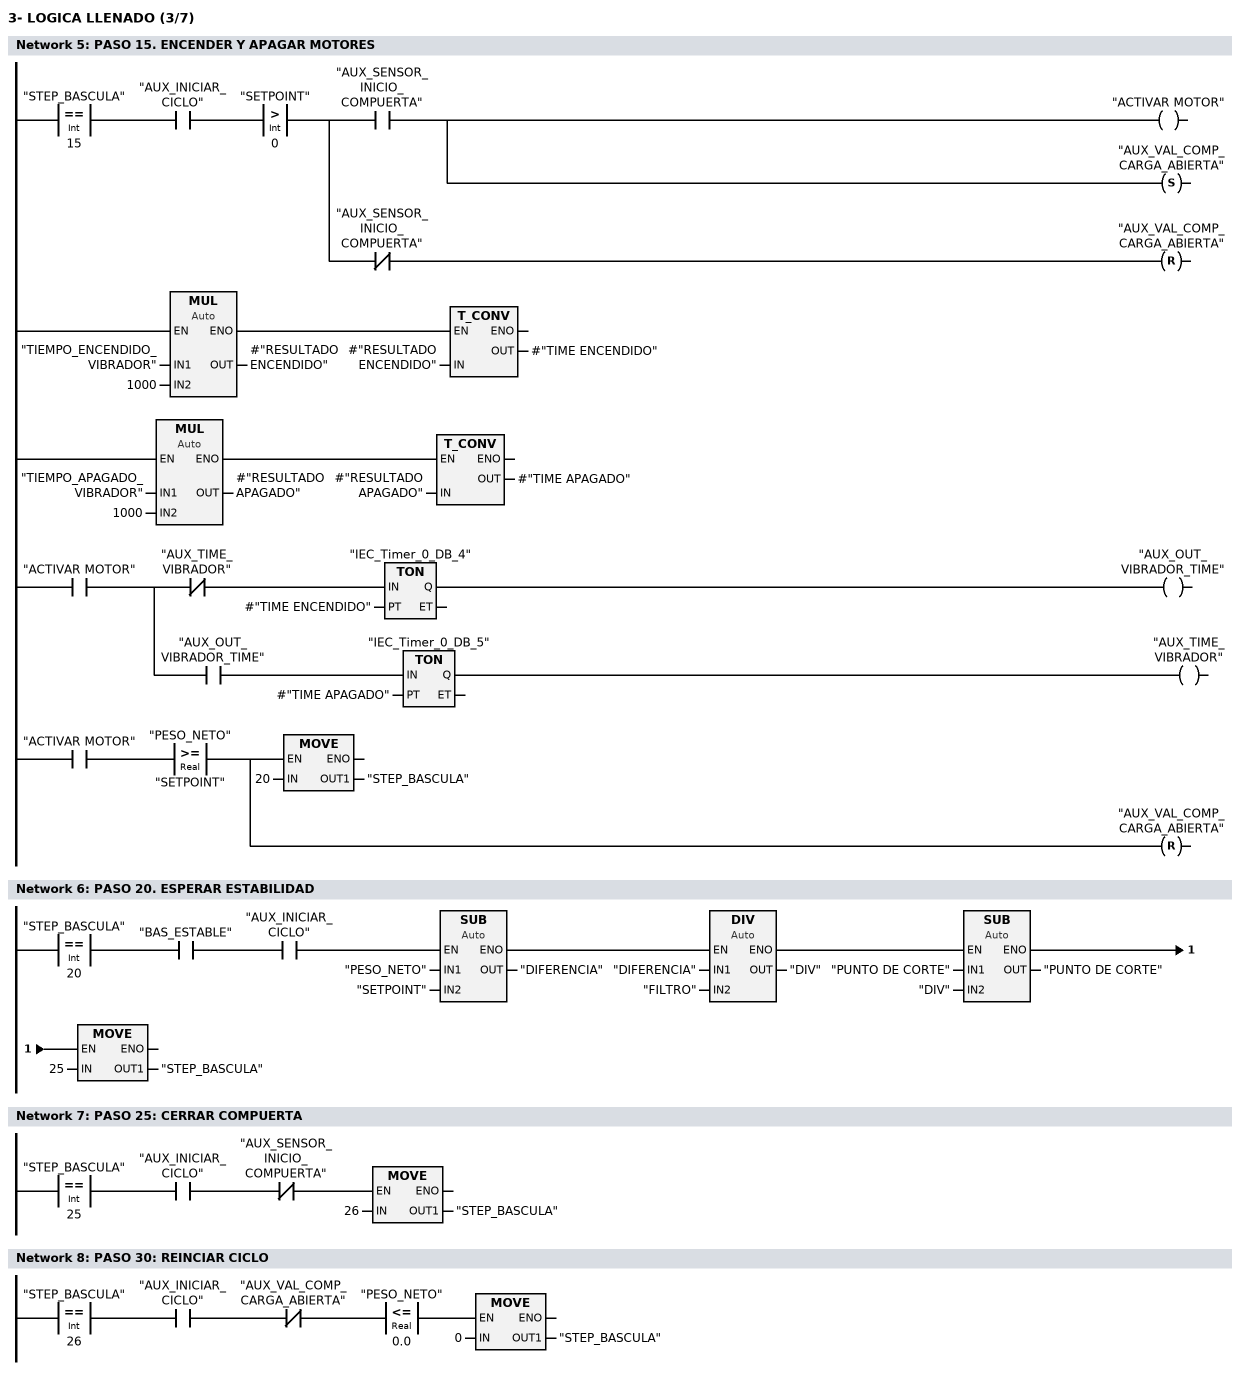
   #_w1 := ("STEP_BASCULA" = 15) AND "AUX_INICIAR_CICLO" AND ("SETPOINT" > 0);
   "ACTIVAR MOTOR" := #_w1 AND "AUX_SENSOR_INICIO_COMPUERTA";
   IF "ACTIVAR MOTOR" THEN "AUX_VAL_COMP_CARGA_ABIERTA" := TRUE; END_IF;
   IF #_w1 AND NOT "AUX_SENSOR_INICIO_COMPUERTA" THEN "AUX_VAL_COMP_CARGA_ABIERTA" := FALSE; END_IF;
   #"RESULTADO ENCENDIDO" := "TIEMPO_ENCENDIDO_VIBRADOR" * 1000;
   #"TIME ENCENDIDO" := T_CONV(IN := #"RESULTADO ENCENDIDO");
   #"RESULTADO APAGADO" := "TIEMPO_APAGADO_VIBRADOR" * 1000;
   #"TIME APAGADO" := T_CONV(IN := #"RESULTADO APAGADO");
   "IEC_Timer_0_DB_4".TON(IN := "ACTIVAR MOTOR" AND NOT "AUX_TIME_VIBRADOR", PT := #"TIME ENCENDIDO");
   "AUX_OUT_VIBRADOR_TIME" := "IEC_Timer_0_DB_4".Q;
   "IEC_Timer_0_DB_5".TON(IN := "ACTIVAR MOTOR" AND "AUX_OUT_VIBRADOR_TIME", PT := #"TIME APAGADO");
   "AUX_TIME_VIBRADOR" := "IEC_Timer_0_DB_5".Q;
   IF "ACTIVAR MOTOR" AND ("PESO_NETO" >= "SETPOINT") THEN
       "STEP_BASCULA" := 20;
       "AUX_VAL_COMP_CARGA_ABIERTA" := FALSE;
   END_IF;
END_REGION

REGION Network 6: PASO 20. ESPERAR ESTABILIDAD
   RUNG wire#powerrail
      { S7_Templates := "SrcType := Int" } EQ_Contact(in1 := "STEP_BASCULA", in2 := 20)
      Contact( "BAS_ESTABLE" )
      Contact( "AUX_INICIAR_CICLO" )
      Sub(in1 := "PESO_NETO", in2 := "SETPOINT", out => "DIFERENCIA")
      Div(in1 := "DIFERENCIA", in2 := "FILTRO", out => "DIV")
      Sub(in1 := "PUNTO DE CORTE", in2 := "DIV", out => "PUNTO DE CORTE")
      Move(in := 25, out1 => "STEP_BASCULA")
   END_RUNG
   // the same network as SCL:
   IF ("STEP_BASCULA" = 20) AND "BAS_ESTABLE" AND "AUX_INICIAR_CICLO" THEN
       "DIFERENCIA" := "PESO_NETO" - "SETPOINT";
       "DIV" := "DIFERENCIA" / "FILTRO";
       "PUNTO DE CORTE" := "PUNTO DE CORTE" - "DIV";
       "STEP_BASCULA" := 25;
   END_IF;
END_REGION

REGION Network 7: PASO 25: CERRAR COMPUERTA
   RUNG wire#powerrail
      { S7_Templates := "SrcType := Int" } EQ_Contact(in1 := "STEP_BASCULA", in2 := 25)
      Contact( "AUX_INICIAR_CICLO" )
      I_Contact( "AUX_SENSOR_INICIO_COMPUERTA" )
      Move(in := 26, out1 => "STEP_BASCULA")
   END_RUNG
   // the same network as SCL:
   IF ("STEP_BASCULA" = 25) AND "AUX_INICIAR_CICLO" AND NOT "AUX_SENSOR_INICIO_COMPUERTA" THEN
       "STEP_BASCULA" := 26;
   END_IF;
END_REGION

REGION Network 8: PASO 30: REINCIAR CICLO
   RUNG wire#powerrail
      { S7_Templates := "SrcType := Int" } EQ_Contact(in1 := "STEP_BASCULA", in2 := 26)
      Contact( "AUX_INICIAR_CICLO" )
      I_Contact( "AUX_VAL_COMP_CARGA_ABIERTA" )
      { S7_Templates := "SrcType := Real" } LE_Contact(in1 := "PESO_NETO", in2 := 0.0)
      Move(in := 0, out1 => "STEP_BASCULA")
   END_RUNG
   // the same network as SCL:
   IF ("STEP_BASCULA" = 26) AND "AUX_INICIAR_CICLO" AND NOT "AUX_VAL_COMP_CARGA_ABIERTA" AND ("PESO_NETO" <= 0.0) THEN
       "STEP_BASCULA" := 0;
   END_IF;
END_REGION

REGION Network 9: CONTROL MANUAL Y BARRIDO DE MOTOR
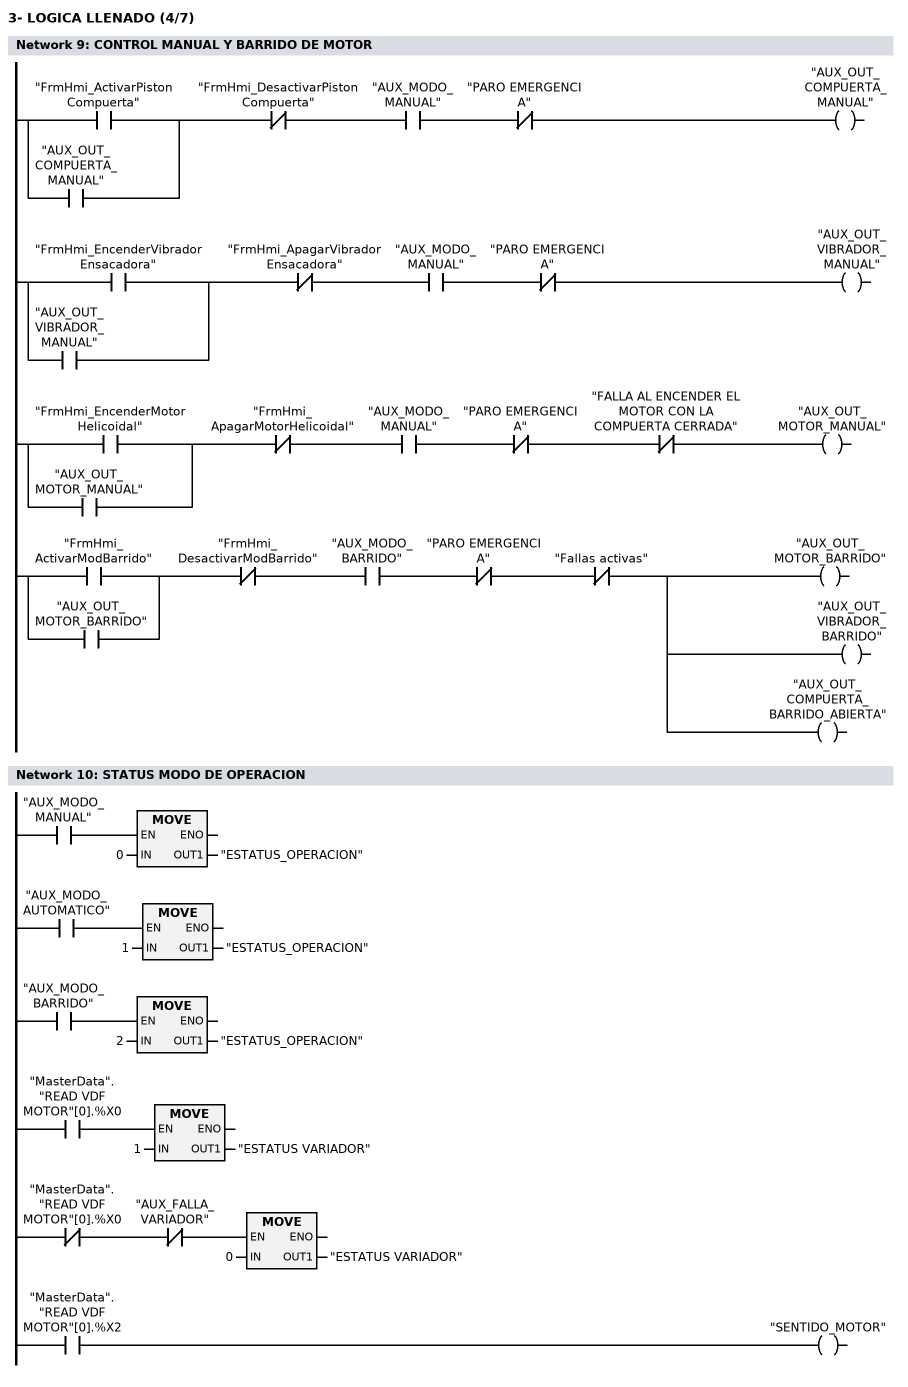
   RUNG wire#powerrail
      Contact( "FrmHmi_ActivarPistonCompuerta" )
      wire#w1
      I_Contact( "FrmHmi_DesactivarPistonCompuerta" )
      Contact( "AUX_MODO_MANUAL" )
      I_Contact( "PARO EMERGENCIA" )
      Coil( "AUX_OUT_COMPUERTA_MANUAL" )
   END_RUNG
   RUNG wire#powerrail
      Contact( "AUX_OUT_COMPUERTA_MANUAL" )
   END_RUNG wire#w1
   RUNG wire#powerrail
      Contact( "FrmHmi_EncenderVibradorEnsacadora" )
      wire#w2
      I_Contact( "FrmHmi_ApagarVibradorEnsacadora" )
      Contact( "AUX_MODO_MANUAL" )
      I_Contact( "PARO EMERGENCIA" )
      Coil( "AUX_OUT_VIBRADOR_MANUAL" )
   END_RUNG
   RUNG wire#powerrail
      Contact( "AUX_OUT_VIBRADOR_MANUAL" )
   END_RUNG wire#w2
   RUNG wire#powerrail
      Contact( "FrmHmi_EncenderMotorHelicoidal" )
      wire#w3
      I_Contact( "FrmHmi_ApagarMotorHelicoidal" )
      Contact( "AUX_MODO_MANUAL" )
      I_Contact( "PARO EMERGENCIA" )
      I_Contact( "FALLA AL ENCENDER EL MOTOR CON LA COMPUERTA CERRADA" )
      Coil( "AUX_OUT_MOTOR_MANUAL" )
   END_RUNG
   RUNG wire#powerrail
      Contact( "AUX_OUT_MOTOR_MANUAL" )
   END_RUNG wire#w3
   RUNG wire#powerrail
      Contact( "FrmHmi_ActivarModBarrido" )
      wire#w4
      I_Contact( "FrmHmi_DesactivarModBarrido" )
      Contact( "AUX_MODO_BARRIDO" )
      I_Contact( "PARO EMERGENCIA" )
      I_Contact( "Fallas activas" )
      wire#w5
      Coil( "AUX_OUT_MOTOR_BARRIDO" )
   END_RUNG
   RUNG wire#powerrail
      Contact( "AUX_OUT_MOTOR_BARRIDO" )
   END_RUNG wire#w4
   RUNG wire#w5
      Coil( "AUX_OUT_VIBRADOR_BARRIDO" )
   END_RUNG
   RUNG wire#w5
      Coil( "AUX_OUT_COMPUERTA_BARRIDO_ABIERTA" )
   END_RUNG
   // the same network as SCL:
   "AUX_OUT_COMPUERTA_MANUAL" := ("FrmHmi_ActivarPistonCompuerta" OR "AUX_OUT_COMPUERTA_MANUAL") AND NOT "FrmHmi_DesactivarPistonCompuerta" AND "AUX_MODO_MANUAL" AND NOT "PARO EMERGENCIA";
   "AUX_OUT_VIBRADOR_MANUAL" := ("FrmHmi_EncenderVibradorEnsacadora" OR "AUX_OUT_VIBRADOR_MANUAL") AND NOT "FrmHmi_ApagarVibradorEnsacadora" AND "AUX_MODO_MANUAL" AND NOT "PARO EMERGENCIA";
   "AUX_OUT_MOTOR_MANUAL" := ("FrmHmi_EncenderMotorHelicoidal" OR "AUX_OUT_MOTOR_MANUAL") AND NOT "FrmHmi_ApagarMotorHelicoidal" AND "AUX_MODO_MANUAL" AND NOT "PARO EMERGENCIA" AND NOT "FALLA AL ENCENDER EL MOTOR CON LA COMPUERTA CERRADA";
   "AUX_OUT_MOTOR_BARRIDO" := ("FrmHmi_ActivarModBarrido" OR "AUX_OUT_MOTOR_BARRIDO") AND NOT "FrmHmi_DesactivarModBarrido" AND "AUX_MODO_BARRIDO" AND NOT "PARO EMERGENCIA" AND NOT "Fallas activas";
   "AUX_OUT_VIBRADOR_BARRIDO" := "AUX_OUT_MOTOR_BARRIDO";
   "AUX_OUT_COMPUERTA_BARRIDO_ABIERTA" := "AUX_OUT_MOTOR_BARRIDO";
END_REGION

REGION Network 10: STATUS MODO DE OPERACION
   RUNG wire#powerrail
      Contact( "AUX_MODO_MANUAL" )
      Move(in := 0, out1 => "ESTATUS_OPERACION")
   END_RUNG
   RUNG wire#powerrail
      Contact( "AUX_MODO_AUTOMATICO" )
      Move(in := 1, out1 => "ESTATUS_OPERACION")
   END_RUNG
   RUNG wire#powerrail
      Contact( "AUX_MODO_BARRIDO" )
      Move(in := 2, out1 => "ESTATUS_OPERACION")
   END_RUNG
   RUNG wire#powerrail
      Contact( "MasterData"."READ VDF MOTOR"[0].%X0 )
      Move(in := 1, out1 => "ESTATUS VARIADOR")
   END_RUNG
   RUNG wire#powerrail
      I_Contact( "MasterData"."READ VDF MOTOR"[0].%X0 )
      I_Contact( "AUX_FALLA_VARIADOR" )
      Move(in := 0, out1 => "ESTATUS VARIADOR")
   END_RUNG
   RUNG wire#powerrail
      Contact( "MasterData"."READ VDF MOTOR"[0].%X2 )
      Coil( "SENTIDO_MOTOR" )
   END_RUNG
   // the same network as SCL:
   IF "AUX_MODO_MANUAL" THEN "ESTATUS_OPERACION" := 0; END_IF;
   IF "AUX_MODO_AUTOMATICO" THEN "ESTATUS_OPERACION" := 1; END_IF;
   IF "AUX_MODO_BARRIDO" THEN "ESTATUS_OPERACION" := 2; END_IF;
   IF "MasterData"."READ VDF MOTOR"[0].%X0 THEN "ESTATUS VARIADOR" := 1; END_IF;
   IF NOT "MasterData"."READ VDF MOTOR"[0].%X0 AND NOT "AUX_FALLA_VARIADOR" THEN
       "ESTATUS VARIADOR" := 0;
   END_IF;
   "SENTIDO_MOTOR" := "MasterData"."READ VDF MOTOR"[0].%X2;
END_REGION

REGION Network 11: FALLAS
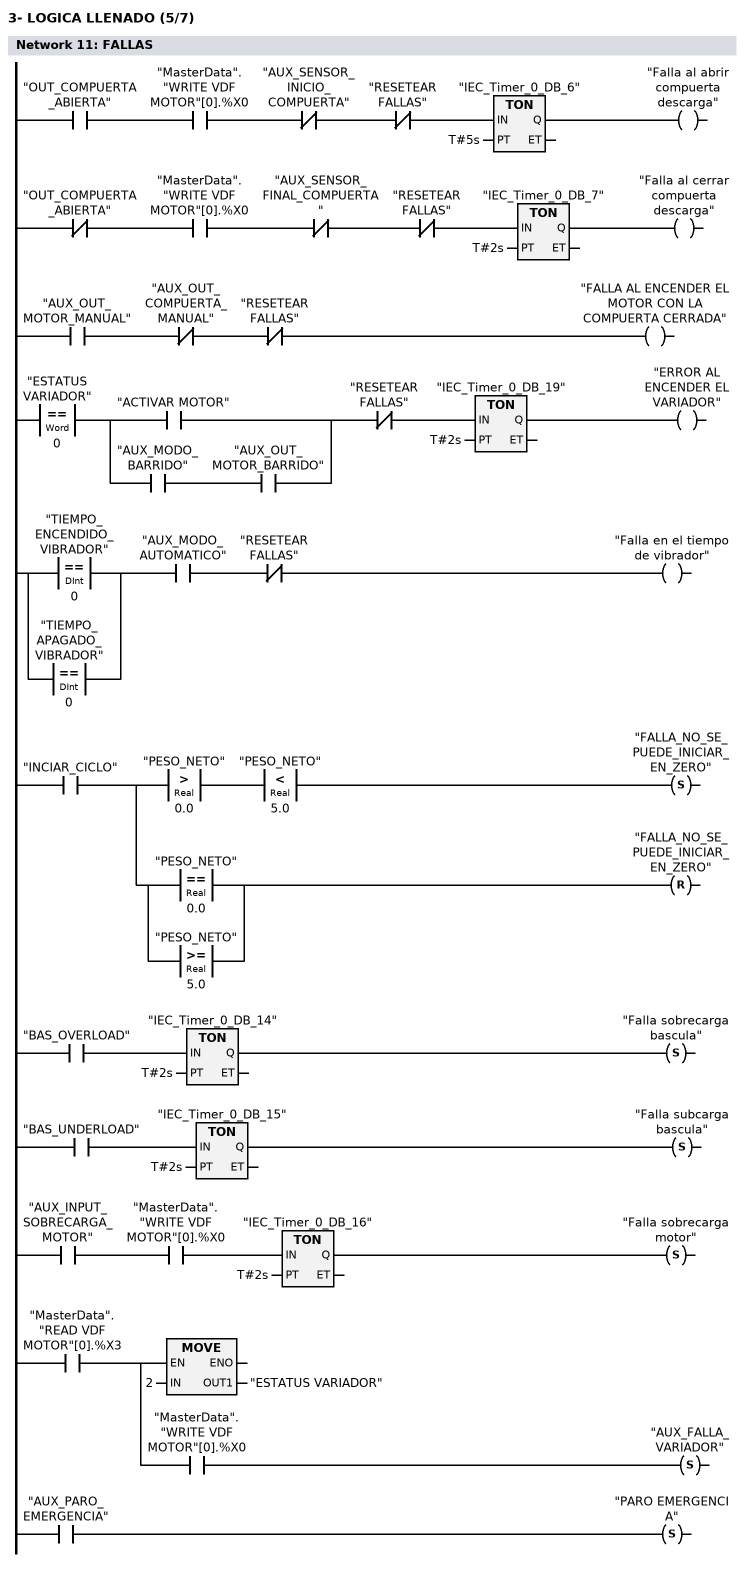
   "IEC_Timer_0_DB_6".TON(IN := "OUT_COMPUERTA_ABIERTA" AND "MasterData"."WRITE VDF MOTOR"[0].%X0 AND NOT "AUX_SENSOR_INICIO_COMPUERTA" AND NOT "RESETEAR FALLAS",
                          PT := T#5s);
   "Falla al abrir compuerta descarga" := "IEC_Timer_0_DB_6".Q;
   "IEC_Timer_0_DB_7".TON(IN := NOT "OUT_COMPUERTA_ABIERTA" AND "MasterData"."WRITE VDF MOTOR"[0].%X0 AND NOT "AUX_SENSOR_FINAL_COMPUERTA" AND NOT "RESETEAR FALLAS",
                          PT := T#2s);
   "Falla al cerrar compuerta descarga" := "IEC_Timer_0_DB_7".Q;
   "FALLA AL ENCENDER EL MOTOR CON LA COMPUERTA CERRADA" := "AUX_OUT_MOTOR_MANUAL" AND NOT "AUX_OUT_COMPUERTA_MANUAL" AND NOT "RESETEAR FALLAS";
   "IEC_Timer_0_DB_19".TON(IN := ("ESTATUS VARIADOR" = 0) AND ("ACTIVAR MOTOR" OR ("AUX_MODO_BARRIDO" AND "AUX_OUT_MOTOR_BARRIDO")) AND NOT "RESETEAR FALLAS",
                           PT := T#2s);
   "ERROR AL ENCENDER EL VARIADOR" := "IEC_Timer_0_DB_19".Q;
   "Falla en el tiempo de vibrador" := (("TIEMPO_ENCENDIDO_VIBRADOR" = 0) OR ("TIEMPO_APAGADO_VIBRADOR" = 0)) AND "AUX_MODO_AUTOMATICO" AND NOT "RESETEAR FALLAS";
   IF "INCIAR_CICLO" AND ("PESO_NETO" > 0.0) AND ("PESO_NETO" < 5.0) THEN
       "FALLA_NO_SE_PUEDE_INICIAR_EN_ZERO" := TRUE;
   END_IF;
   IF "INCIAR_CICLO" AND (("PESO_NETO" = 0.0) OR ("PESO_NETO" >= 5.0)) THEN
       "FALLA_NO_SE_PUEDE_INICIAR_EN_ZERO" := FALSE;
   END_IF;
   "IEC_Timer_0_DB_14".TON(IN := "BAS_OVERLOAD", PT := T#2s);
   IF "IEC_Timer_0_DB_14".Q THEN "Falla sobrecarga bascula" := TRUE; END_IF;
   "IEC_Timer_0_DB_15".TON(IN := "BAS_UNDERLOAD", PT := T#2s);
   IF "IEC_Timer_0_DB_15".Q THEN "Falla subcarga bascula" := TRUE; END_IF;
   "IEC_Timer_0_DB_16".TON(IN := "AUX_INPUT_SOBRECARGA_MOTOR" AND "MasterData"."WRITE VDF MOTOR"[0].%X0,
                           PT := T#2s);
   IF "IEC_Timer_0_DB_16".Q THEN "Falla sobrecarga motor" := TRUE; END_IF;
   IF "MasterData"."READ VDF MOTOR"[0].%X3 THEN "ESTATUS VARIADOR" := 2; END_IF;
   IF "MasterData"."READ VDF MOTOR"[0].%X3 AND "MasterData"."WRITE VDF MOTOR"[0].%X0 THEN
       "AUX_FALLA_VARIADOR" := TRUE;
   END_IF;
   IF "AUX_PARO_EMERGENCIA" THEN "PARO EMERGENCIA" := TRUE; END_IF;
END_REGION

REGION Network 12: FALLAS ACTIVAS
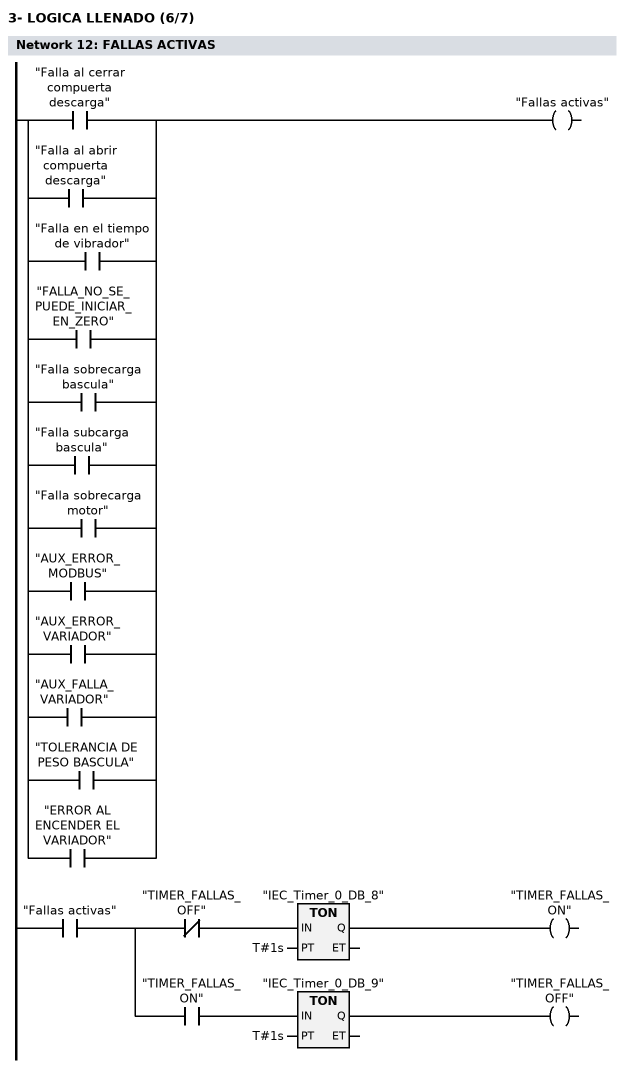
   "Fallas activas" := "Falla al cerrar compuerta descarga" OR "Falla al abrir compuerta descarga" OR "Falla en el tiempo de vibrador" OR "FALLA_NO_SE_PUEDE_INICIAR_EN_ZERO" OR "Falla sobrecarga bascula" OR "Falla subcarga bascula" OR "Falla sobrecarga motor" OR "AUX_ERROR_MODBUS" OR "AUX_ERROR_VARIADOR" OR "AUX_FALLA_VARIADOR" OR "TOLERANCIA DE PESO BASCULA" OR "ERROR AL ENCENDER EL VARIADOR";
   "IEC_Timer_0_DB_8".TON(IN := "Fallas activas" AND NOT "TIMER_FALLAS_OFF", PT := T#1s);
   "TIMER_FALLAS_ON" := "IEC_Timer_0_DB_8".Q;
   "IEC_Timer_0_DB_9".TON(IN := "Fallas activas" AND "TIMER_FALLAS_ON", PT := T#1s);
   "TIMER_FALLAS_OFF" := "IEC_Timer_0_DB_9".Q;
END_REGION

REGION Network 13: RESET SET FALLAS
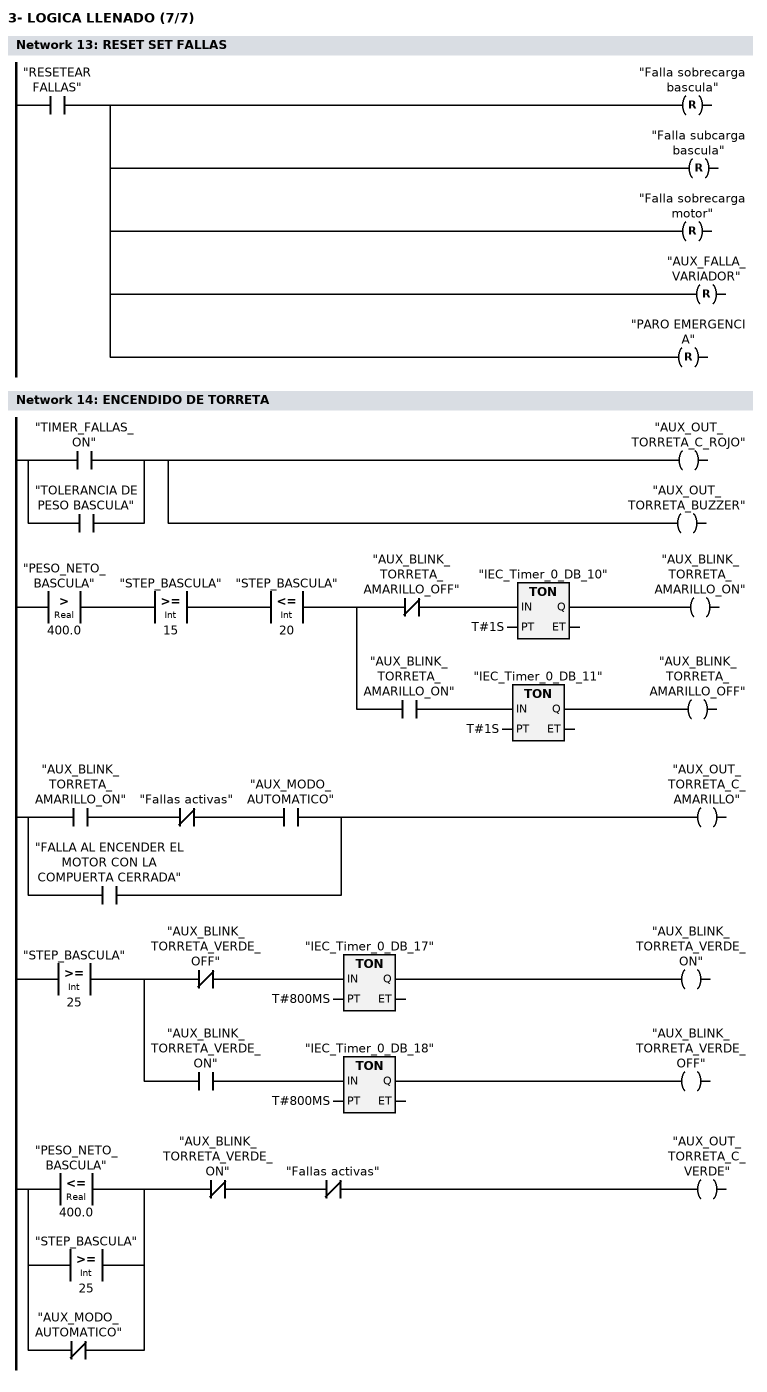
   RUNG wire#powerrail
      Contact( "RESETEAR FALLAS" )
      wire#w1
      R_Coil( "Falla sobrecarga bascula" )
   END_RUNG
   RUNG wire#w1
      R_Coil( "Falla subcarga bascula" )
   END_RUNG
   RUNG wire#w1
      R_Coil( "Falla sobrecarga motor" )
   END_RUNG
   RUNG wire#w1
      R_Coil( "AUX_FALLA_VARIADOR" )
   END_RUNG
   RUNG wire#w1
      R_Coil( "PARO EMERGENCIA" )
   END_RUNG
   // the same network as SCL:
   IF "RESETEAR FALLAS" THEN
       "Falla sobrecarga bascula" := FALSE;
       "Falla subcarga bascula" := FALSE;
       "Falla sobrecarga motor" := FALSE;
       "AUX_FALLA_VARIADOR" := FALSE;
       "PARO EMERGENCIA" := FALSE;
   END_IF;
END_REGION

REGION Network 14: ENCENDIDO DE TORRETA
   "AUX_OUT_TORRETA_C_ROJO" := "TIMER_FALLAS_ON" OR "TOLERANCIA DE PESO BASCULA";
   "AUX_OUT_TORRETA_BUZZER" := "AUX_OUT_TORRETA_C_ROJO";
   #_w1 := ("PESO_NETO_BASCULA" > 400.0) AND ("STEP_BASCULA" >= 15) AND ("STEP_BASCULA" <= 20);
   "IEC_Timer_0_DB_10".TON(IN := #_w1 AND NOT "AUX_BLINK_TORRETA_AMARILLO_OFF", PT := T#1S);
   "AUX_BLINK_TORRETA_AMARILLO_ON" := "IEC_Timer_0_DB_10".Q;
   "IEC_Timer_0_DB_11".TON(IN := #_w1 AND "AUX_BLINK_TORRETA_AMARILLO_ON", PT := T#1S);
   "AUX_BLINK_TORRETA_AMARILLO_OFF" := "IEC_Timer_0_DB_11".Q;
   "AUX_OUT_TORRETA_C_AMARILLO" := ("AUX_BLINK_TORRETA_AMARILLO_ON" AND NOT "Fallas activas" AND "AUX_MODO_AUTOMATICO") OR "FALLA AL ENCENDER EL MOTOR CON LA COMPUERTA CERRADA";
   #_w2 := "STEP_BASCULA" >= 25;
   "IEC_Timer_0_DB_17".TON(IN := #_w2 AND NOT "AUX_BLINK_TORRETA_VERDE_OFF", PT := T#800MS);
   "AUX_BLINK_TORRETA_VERDE_ON" := "IEC_Timer_0_DB_17".Q;
   "IEC_Timer_0_DB_18".TON(IN := #_w2 AND "AUX_BLINK_TORRETA_VERDE_ON", PT := T#800MS);
   "AUX_BLINK_TORRETA_VERDE_OFF" := "IEC_Timer_0_DB_18".Q;
   "AUX_OUT_TORRETA_C_VERDE" := (("PESO_NETO_BASCULA" <= 400.0) OR ("STEP_BASCULA" >= 25) OR NOT "AUX_MODO_AUTOMATICO") AND NOT "AUX_BLINK_TORRETA_VERDE_ON" AND NOT "Fallas activas";
END_REGION
END_ORGANIZATION_BLOCK

ORGANIZATION_BLOCK "4- SALIDAS"   // OB125, LAD, ProgramCycle
{ S7_Optimized_Access := 'TRUE' }
VERSION : 0.1
   VAR_INPUT
      Initial_Call : Bool;
      Remanence : Bool;
   END_VAR
   VAR_TEMP
      INHABILITADO : Bool;
      OUT : Bool;
      available : Bool;
   END_VAR
BEGIN

REGION Network 1: OUT VIBRADOR , VARIADOR Y COMPUERTA
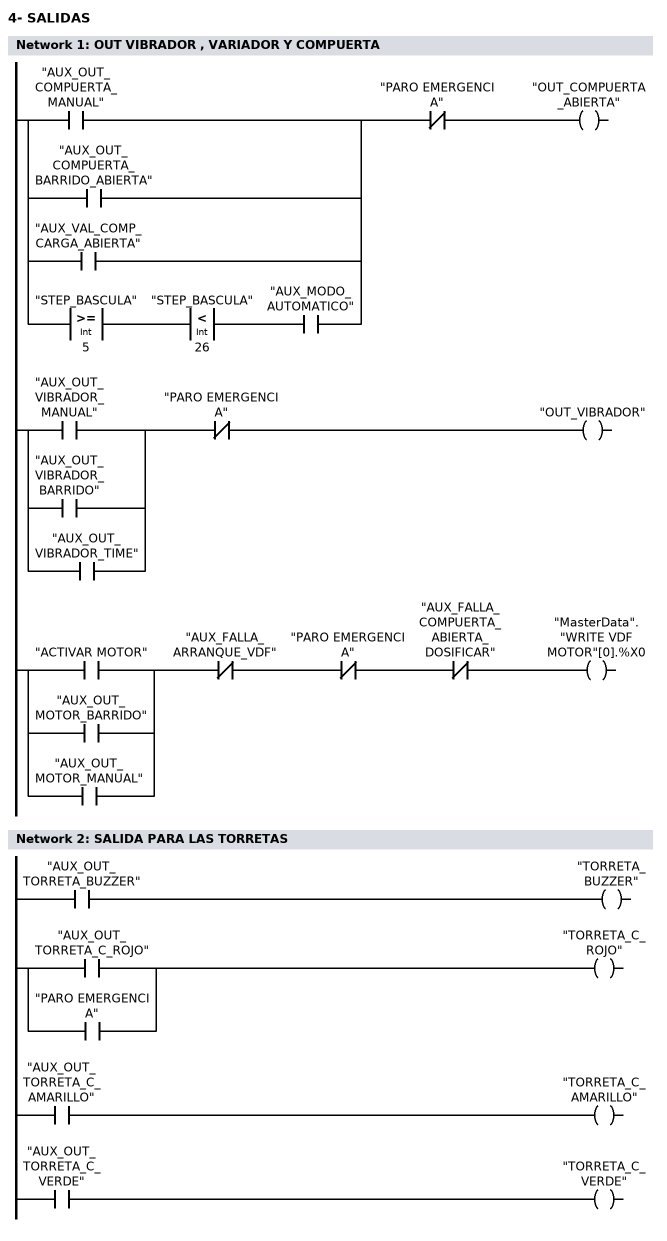
   RUNG wire#powerrail
      Contact( "AUX_OUT_COMPUERTA_MANUAL" )
      wire#w1
      I_Contact( "PARO EMERGENCIA" )
      Coil( "OUT_COMPUERTA_ABIERTA" )
   END_RUNG
   RUNG wire#powerrail
      Contact( "AUX_OUT_COMPUERTA_BARRIDO_ABIERTA" )
   END_RUNG wire#w1
   RUNG wire#powerrail
      Contact( "AUX_VAL_COMP_CARGA_ABIERTA" )
   END_RUNG wire#w1
   RUNG wire#powerrail
      { S7_Templates := "SrcType := Int" } GE_Contact(in1 := "STEP_BASCULA", in2 := 5)
      { S7_Templates := "SrcType := Int" } LT_Contact(in1 := "STEP_BASCULA", in2 := 26)
      Contact( "AUX_MODO_AUTOMATICO" )
   END_RUNG wire#w1
   RUNG wire#powerrail
      Contact( "AUX_OUT_VIBRADOR_MANUAL" )
      wire#w2
      I_Contact( "PARO EMERGENCIA" )
      Coil( "OUT_VIBRADOR" )
   END_RUNG
   RUNG wire#powerrail
      Contact( "AUX_OUT_VIBRADOR_BARRIDO" )
   END_RUNG wire#w2
   RUNG wire#powerrail
      Contact( "AUX_OUT_VIBRADOR_TIME" )
   END_RUNG wire#w2
   RUNG wire#powerrail
      Contact( "ACTIVAR MOTOR" )
      wire#w3
      I_Contact( "AUX_FALLA_ARRANQUE_VDF" )
      I_Contact( "PARO EMERGENCIA" )
      I_Contact( "AUX_FALLA_COMPUERTA_ABIERTA_DOSIFICAR" )
      Coil( "MasterData"."WRITE VDF MOTOR"[0].%X0 )
   END_RUNG
   RUNG wire#powerrail
      Contact( "AUX_OUT_MOTOR_BARRIDO" )
   END_RUNG wire#w3
   RUNG wire#powerrail
      Contact( "AUX_OUT_MOTOR_MANUAL" )
   END_RUNG wire#w3
   // the same network as SCL:
   "OUT_COMPUERTA_ABIERTA" := ("AUX_OUT_COMPUERTA_MANUAL" OR "AUX_OUT_COMPUERTA_BARRIDO_ABIERTA" OR "AUX_VAL_COMP_CARGA_ABIERTA" OR (("STEP_BASCULA" >= 5) AND ("STEP_BASCULA" < 26) AND "AUX_MODO_AUTOMATICO")) AND NOT "PARO EMERGENCIA";
   "OUT_VIBRADOR" := ("AUX_OUT_VIBRADOR_MANUAL" OR "AUX_OUT_VIBRADOR_BARRIDO" OR "AUX_OUT_VIBRADOR_TIME") AND NOT "PARO EMERGENCIA";
   "MasterData"."WRITE VDF MOTOR"[0].%X0 := ("ACTIVAR MOTOR" OR "AUX_OUT_MOTOR_BARRIDO" OR "AUX_OUT_MOTOR_MANUAL") AND NOT "AUX_FALLA_ARRANQUE_VDF" AND NOT "PARO EMERGENCIA" AND NOT "AUX_FALLA_COMPUERTA_ABIERTA_DOSIFICAR";
END_REGION

REGION Network 2: SALIDA PARA LAS TORRETAS
   RUNG wire#powerrail
      Contact( "AUX_OUT_TORRETA_BUZZER" )
      Coil( "TORRETA_BUZZER" )
   END_RUNG
   RUNG wire#powerrail
      Contact( "AUX_OUT_TORRETA_C_ROJO" )
      wire#w1
      Coil( "TORRETA_C_ROJO" )
   END_RUNG
   RUNG wire#powerrail
      Contact( "PARO EMERGENCIA" )
   END_RUNG wire#w1
   RUNG wire#powerrail
      Contact( "AUX_OUT_TORRETA_C_AMARILLO" )
      Coil( "TORRETA_C_AMARILLO" )
   END_RUNG
   RUNG wire#powerrail
      Contact( "AUX_OUT_TORRETA_C_VERDE" )
      Coil( "TORRETA_C_VERDE" )
   END_RUNG
   // the same network as SCL:
   "TORRETA_BUZZER" := "AUX_OUT_TORRETA_BUZZER";
   "TORRETA_C_ROJO" := "AUX_OUT_TORRETA_C_ROJO" OR "PARO EMERGENCIA";
   "TORRETA_C_AMARILLO" := "AUX_OUT_TORRETA_C_AMARILLO";
   "TORRETA_C_VERDE" := "AUX_OUT_TORRETA_C_VERDE";
END_REGION
END_ORGANIZATION_BLOCK

ORGANIZATION_BLOCK "5- CALIBRACION"   // OB126, LAD, ProgramCycle
{ S7_Optimized_Access := 'TRUE' }
VERSION : 0.1
   VAR_INPUT
      Initial_Call : Bool;
      Remanence : Bool;
   END_VAR
   VAR_TEMP
      AVAILABLE : Bool;
   END_VAR
BEGIN

REGION Network 1: VER CALIBRACION EN HMI
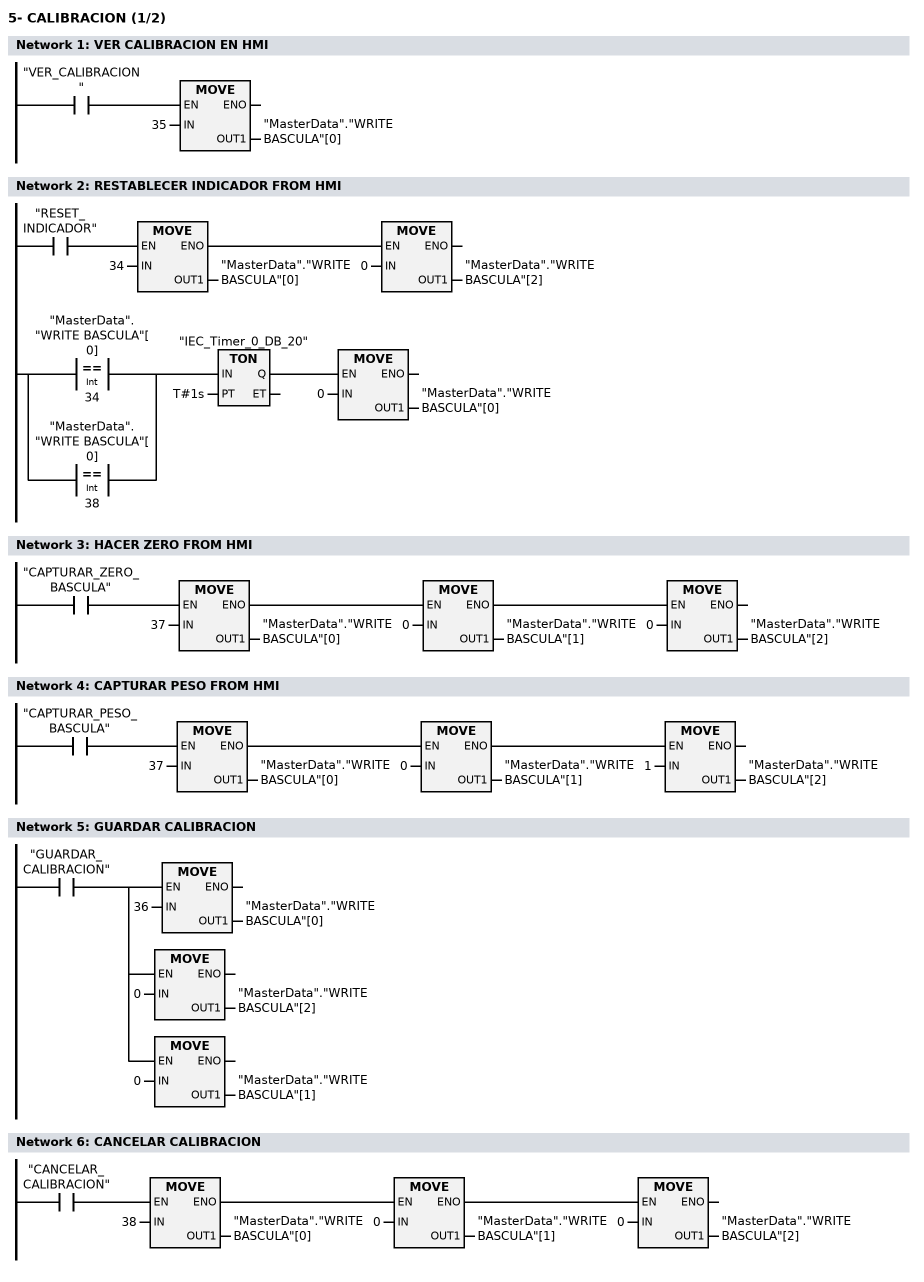
   RUNG wire#powerrail
      Contact( "VER_CALIBRACION" )
      Move(in := 35, out1 => "MasterData"."WRITE BASCULA"[0])
   END_RUNG
   // the same network as SCL:
   IF "VER_CALIBRACION" THEN "MasterData"."WRITE BASCULA"[0] := 35; END_IF;
END_REGION

REGION Network 2: RESTABLECER INDICADOR FROM HMI
   IF "RESET_INDICADOR" THEN
       "MasterData"."WRITE BASCULA"[0] := 34;
       "MasterData"."WRITE BASCULA"[2] := 0;
   END_IF;
   "IEC_Timer_0_DB_20".TON(IN := ("MasterData"."WRITE BASCULA"[0] = 34) OR ("MasterData"."WRITE BASCULA"[0] = 38),
                           PT := T#1s);
   IF "IEC_Timer_0_DB_20".Q THEN "MasterData"."WRITE BASCULA"[0] := 0; END_IF;
END_REGION

REGION Network 3: HACER ZERO FROM HMI
   RUNG wire#powerrail
      Contact( "CAPTURAR_ZERO_BASCULA" )
      Move(in := 37, out1 => "MasterData"."WRITE BASCULA"[0])
      Move(in := 0, out1 => "MasterData"."WRITE BASCULA"[1])
      Move(in := 0, out1 => "MasterData"."WRITE BASCULA"[2])
   END_RUNG
   // the same network as SCL:
   IF "CAPTURAR_ZERO_BASCULA" THEN
       "MasterData"."WRITE BASCULA"[0] := 37;
       "MasterData"."WRITE BASCULA"[1] := 0;
       "MasterData"."WRITE BASCULA"[2] := 0;
   END_IF;
END_REGION

REGION Network 4: CAPTURAR PESO FROM HMI
   RUNG wire#powerrail
      Contact( "CAPTURAR_PESO_BASCULA" )
      Move(in := 37, out1 => "MasterData"."WRITE BASCULA"[0])
      Move(in := 0, out1 => "MasterData"."WRITE BASCULA"[1])
      Move(in := 1, out1 => "MasterData"."WRITE BASCULA"[2])
   END_RUNG
   // the same network as SCL:
   IF "CAPTURAR_PESO_BASCULA" THEN
       "MasterData"."WRITE BASCULA"[0] := 37;
       "MasterData"."WRITE BASCULA"[1] := 0;
       "MasterData"."WRITE BASCULA"[2] := 1;
   END_IF;
END_REGION

REGION Network 5: GUARDAR CALIBRACION
   RUNG wire#powerrail
      Contact( "GUARDAR_CALIBRACION" )
      wire#w1
      Move(in := 36, out1 => "MasterData"."WRITE BASCULA"[0])
   END_RUNG
   RUNG wire#w1
      Move(in := 0, out1 => "MasterData"."WRITE BASCULA"[2])
   END_RUNG
   RUNG wire#w1
      Move(in := 0, out1 => "MasterData"."WRITE BASCULA"[1])
   END_RUNG
   // the same network as SCL:
   IF "GUARDAR_CALIBRACION" THEN
       "MasterData"."WRITE BASCULA"[0] := 36;
       "MasterData"."WRITE BASCULA"[2] := 0;
       "MasterData"."WRITE BASCULA"[1] := 0;
   END_IF;
END_REGION

REGION Network 6: CANCELAR CALIBRACION
   RUNG wire#powerrail
      Contact( "CANCELAR_CALIBRACION" )
      Move(in := 38, out1 => "MasterData"."WRITE BASCULA"[0])
      Move(in := 0, out1 => "MasterData"."WRITE BASCULA"[1])
      Move(in := 0, out1 => "MasterData"."WRITE BASCULA"[2])
   END_RUNG
   // the same network as SCL:
   IF "CANCELAR_CALIBRACION" THEN
       "MasterData"."WRITE BASCULA"[0] := 38;
       "MasterData"."WRITE BASCULA"[1] := 0;
       "MasterData"."WRITE BASCULA"[2] := 0;
   END_IF;
END_REGION

REGION Network 7: CONFIRMAR PESO A CALIBRAR
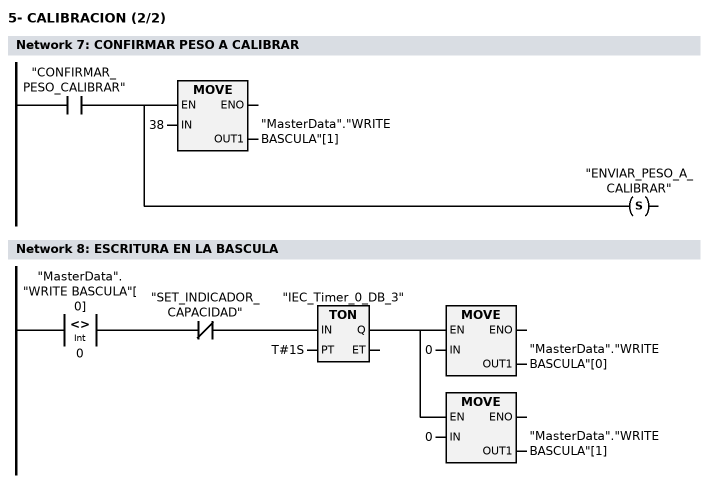
   RUNG wire#powerrail
      Contact( "CONFIRMAR_PESO_CALIBRAR" )
      wire#w1
      Move(in := 38, out1 => "MasterData"."WRITE BASCULA"[1])
   END_RUNG
   RUNG wire#w1
      S_Coil( "ENVIAR_PESO_A_CALIBRAR" )
   END_RUNG
   // the same network as SCL:
   IF "CONFIRMAR_PESO_CALIBRAR" THEN
       "MasterData"."WRITE BASCULA"[1] := 38;
       "ENVIAR_PESO_A_CALIBRAR" := TRUE;
   END_IF;
END_REGION

REGION Network 8: ESCRITURA EN LA BASCULA
   "IEC_Timer_0_DB_3".TON(IN := ("MasterData"."WRITE BASCULA"[0] <> 0) AND NOT "SET_INDICADOR_CAPACIDAD",
                          PT := T#1S);
   IF "IEC_Timer_0_DB_3".Q THEN
       "MasterData"."WRITE BASCULA"[0] := 0;
       "MasterData"."WRITE BASCULA"[1] := 0;
   END_IF;
END_REGION
END_ORGANIZATION_BLOCK

ORGANIZATION_BLOCK "6- CELDAS"   // OB128, LAD, ProgramCycle
TITLE = "Main Program Sweep (Cycle)"
{ S7_Optimized_Access := 'TRUE' }
VERSION : 0.1
   VAR_INPUT
      Initial_Call : Bool;   // Initial call of this OB
      Remanence : Bool;   // =True, if remanent data are available
   END_VAR
   VAR_TEMP
      RESULTADO_SUMA_CELDAS : DInt;
      CONVERTIR_A_REAL : LReal;
      RESTA_AMPERAJE : Real;
      RESTA_CELDAS : Real;
      RESULTADO_DIVISION : Real;
      RESULTADO_MUL : Real;
      RESULTADO_FINAL : Real;
      "RESULTADO EN KILOS" : Real;
      SALIDA_NORM_X : Real;
   END_VAR
BEGIN

REGION Network 1: SUMA DE LAS 4 CELDAS Y CONVERTIR A KILOS
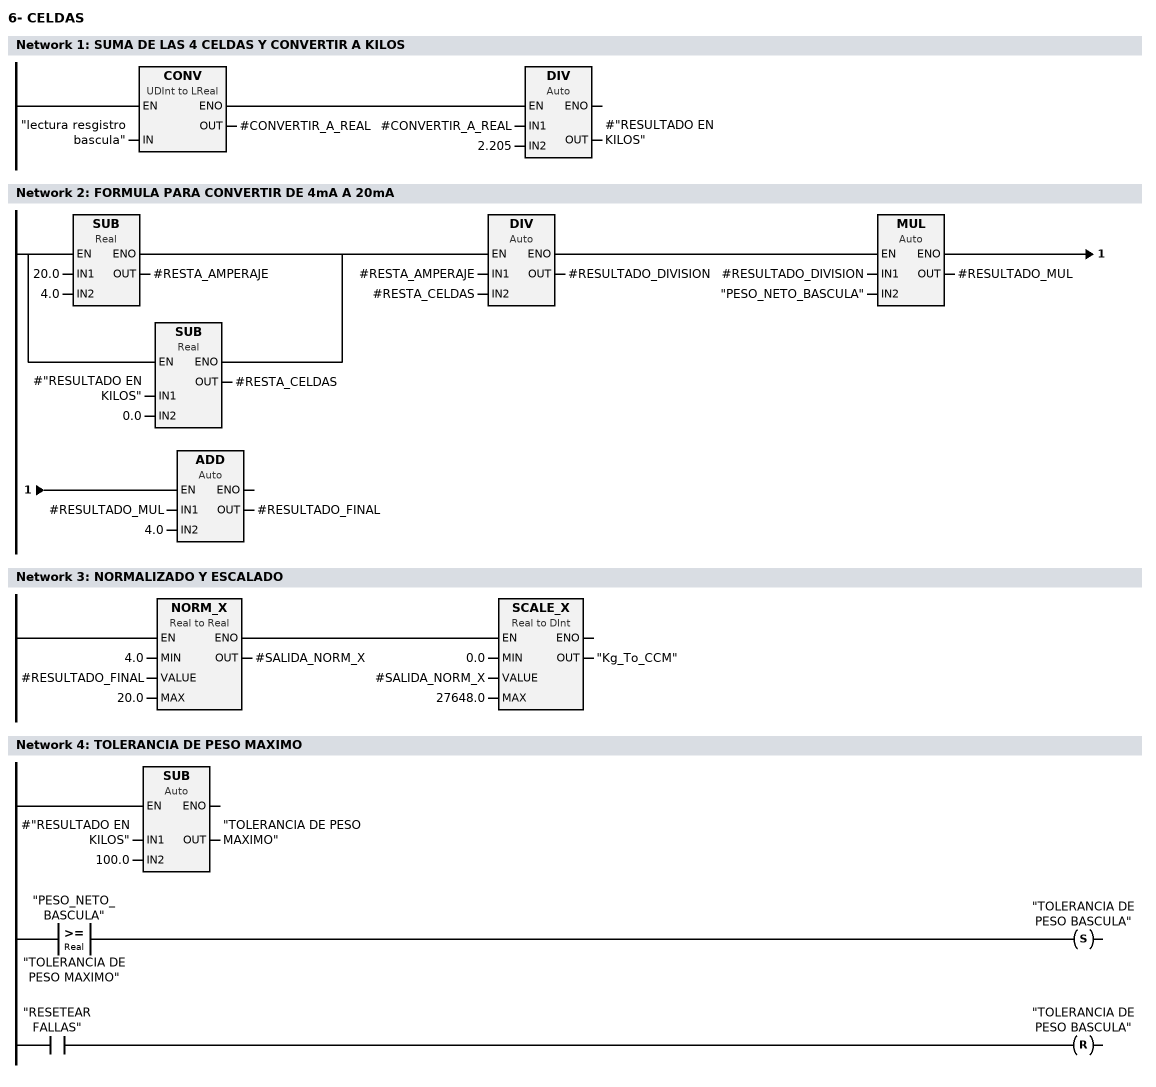
   RUNG wire#powerrail
      { S7_Templates := "[SrcType := UDInt, DestType := LReal]" } Convert(in := "lectura resgistro bascula", out => #CONVERTIR_A_REAL)
      Div(in1 := #CONVERTIR_A_REAL, in2 := 2.205, out => #"RESULTADO EN KILOS")
   END_RUNG
   // the same network as SCL:
   #CONVERTIR_A_REAL := UDINT_TO_LREAL("lectura resgistro bascula");
   #"RESULTADO EN KILOS" := #CONVERTIR_A_REAL / 2.205;
END_REGION

REGION Network 2: FORMULA PARA CONVERTIR DE 4mA A 20mA
   RUNG wire#powerrail
      { S7_Templates := "SrcType := Real" } Sub(in1 := 20.0, in2 := 4.0, out => #RESTA_AMPERAJE)
      wire#w1
      Div(in1 := #RESTA_AMPERAJE, in2 := #RESTA_CELDAS, out => #RESULTADO_DIVISION)
      Mul(in1 := #RESULTADO_DIVISION, in2 := "PESO_NETO_BASCULA", out => #RESULTADO_MUL)
      Add(in1 := #RESULTADO_MUL, in2 := 4.0, out => #RESULTADO_FINAL)
   END_RUNG
   RUNG wire#powerrail
      { S7_Templates := "SrcType := Real" } Sub(in1 := #"RESULTADO EN KILOS", in2 := 0.0, out => #RESTA_CELDAS)
   END_RUNG wire#w1
   // the same network as SCL:
   #RESTA_AMPERAJE := 20.0 - 4.0;
   #RESTA_CELDAS := #"RESULTADO EN KILOS" - 0.0;
   IF TRUE OR TRUE THEN
       #RESULTADO_DIVISION := #RESTA_AMPERAJE / #RESTA_CELDAS;
       #RESULTADO_MUL := #RESULTADO_DIVISION * "PESO_NETO_BASCULA";
       #RESULTADO_FINAL := #RESULTADO_MUL + 4.0;
   END_IF;
END_REGION

REGION Network 3: NORMALIZADO Y ESCALADO
   RUNG wire#powerrail
      { S7_Templates := "[SrcType := Real, DestType := Real]" } Normalize(min := 4.0, value := #RESULTADO_FINAL, max := 20.0, out => #SALIDA_NORM_X)
      { S7_Templates := "[SrcType := Real, DestType := DInt]" } Scale(min := 0.0, value := #SALIDA_NORM_X, max := 27648.0, out => "Kg_To_CCM")
   END_RUNG
   // the same network as SCL:
   #SALIDA_NORM_X := NORM_X(MIN := 4.0, VALUE := #RESULTADO_FINAL, MAX := 20.0);
   "Kg_To_CCM" := SCALE_X(MIN := 0.0, VALUE := #SALIDA_NORM_X, MAX := 27648.0);
END_REGION

REGION Network 4: TOLERANCIA DE PESO MAXIMO
   RUNG wire#powerrail
      Sub(in1 := #"RESULTADO EN KILOS", in2 := 100.0, out => "TOLERANCIA DE PESO MAXIMO")
   END_RUNG
   RUNG wire#powerrail
      { S7_Templates := "SrcType := Real" } GE_Contact(in1 := "PESO_NETO_BASCULA", in2 := "TOLERANCIA DE PESO MAXIMO")
      S_Coil( "TOLERANCIA DE PESO BASCULA" )
   END_RUNG
   RUNG wire#powerrail
      Contact( "RESETEAR FALLAS" )
      R_Coil( "TOLERANCIA DE PESO BASCULA" )
   END_RUNG
   // the same network as SCL:
   "TOLERANCIA DE PESO MAXIMO" := #"RESULTADO EN KILOS" - 100.0;
   IF "PESO_NETO_BASCULA" >= "TOLERANCIA DE PESO MAXIMO" THEN "TOLERANCIA DE PESO BASCULA" := TRUE; END_IF;
   IF "RESETEAR FALLAS" THEN "TOLERANCIA DE PESO BASCULA" := FALSE; END_IF;
END_REGION
END_ORGANIZATION_BLOCK